// TwinCAT 3 PLC project MorpheePanel_PowerSupplyControl
// ProgramVersion: 3.1.4024.0
// libraries:
//   Tc2_Standard, * (Beckhoff Automation GmbH)
//   Tc2_System, * (Beckhoff Automation GmbH)
//   Tc3_Module, * (Beckhoff Automation GmbH)
// project tree:
//   DUTs/ panel302.TcDUT, RxData.TcDUT, TxData.TcDUT
//   GVLs/ GVL.TcGVL, GVL_Constant.TcGVL, GVL_Persistent.TcGVL, Safety_Tags.TcGVL
//   / PlcTask.TcTTO
//   POU/ DeviceManager.TcPOU, EthercatManager.TcPOU, GroupManager.TcPOU, Main.TcPOU, SafetyMgr.TcPOU, SetpointTest.TcPOU
// real-time tasks:
//   TASK PlcTask: cycle T#10ms, priority 20, ADS port 350
// I/O:
//   DEVICE Device 1 (EtherCAT), AmsNetId 5.146.184.42.2.1
//     Term 37 (EK1200) [EK1200-5000 EtherCAT Power supply (2A E-Bus)]
//       Term 2 (EL1819) [EL1819 16Ch. Dig. Input 24V, 10µs]
//       Term 3(EL6695) [EL6695 EtherCAT Bridge terminal (Primary)]
//       Term 4 (EK1521) [EK1521 1 port EtherCAT junction (FX-MultiMode)]
//         Term 5 (EK1501) [EK1501 EtherCAT Coupler (2A E-Bus, FX-MultiMode, ID switch)]
//           Term 6 (EL6070-0033) [EL6070-0033 1Ch. Licence key terminal, individual licences]
//           Term 7 (EL6910) [EL6910, TwinSAFE PLC]
//           Term 8 (EL1819) [EL1819 16Ch. Dig. Input 24V, 10µs]
//           Term 9 (EL1819) [EL1819 16Ch. Dig. Input 24V, 10µs]
//           Term 10 (EL1904) [EL1904, 4 Ch. Safety Input 24V, TwinSAFE]
//             modules: Module 1 (FSOES)
//           Term 11 (EL2809) [EL2809 16Ch. Dig. Output 24V, 0.5A]
//           Term 12 (EL2904) [EL2904, 4 Ch. Safety Output 24V, 0.5A, TwinSAFE]
//             modules: Module 1 (FSOES), Module 2 (DO)
//           Term 13 (EL2798) [EL2798 8Ch. Dig. Output 24V AC/DC, 2A, potential-free]
//           Term 14 (EL9410) [EL9410 E-Bus Power Supplier  (Diagnostics)]
//           Term 15 (EL3174) [EL3174 4Ch. Ana. Input +/-10V Diff., +/-20mA SingleEnded, 16 Bit]
//           Term 52 (EL6751) [EL6751 CANopen Master]
//           Term 53 (EL6751) [EL6751 CANopen Master]
//           Term 54 (EL6751) [EL6751 CANopen Master]
//           Term 20 (EK1122) [EK1122 2 port EtherCAT junction]
//             Box 22 (CX8110 EtherCAT slave) [CX8110 EtherCAT slave]
//       Term 3 (EK1122) [EK1122 2 port EtherCAT junction]
//         Term 48 (EK1100) [EK1100 EtherCAT Coupler (2A E-Bus)]
//           Term 49 (EL1819) [EL1819 16Ch. Dig. Input 24V, 10µs]
//           Term 50 (EL2809) [EL2809 16Ch. Dig. Output 24V, 0.5A]
//           Term 45 (EL1918) [EL1918, 8Ch. Safety Input 24V, TwinSAFE]
//             modules: Module 2 (FSLOGIC)
//           Term 52 (EL2904) [EL2904, 4 Ch. Safety Output 24V, 0.5A, TwinSAFE]
//             modules: Module 1 (FSOES), Module 2 (DO)
//           Term 60 (EL9011) [EL9011 End Terminal]
//         Term 54 (EK1100) [EK1100 EtherCAT Coupler (2A E-Bus)]
//           Term 55 (EL1819) [EL1819 16Ch. Dig. Input 24V, 10µs]
//           Term 56 (EL2809) [EL2809 16Ch. Dig. Output 24V, 0.5A]
//           Term 57 (EL1918) [EL1918, 8Ch. Safety Input 24V, TwinSAFE]
//             modules: Module 1 (FSOE), Module 2 (FSLOGIC)
//           Term 58 (EL2904) [EL2904, 4 Ch. Safety Output 24V, 0.5A, TwinSAFE]
//             modules: Module 1 (FSOES), Module 2 (DO)
//           Term 61 (EL9011) [EL9011 End Terminal]
//   DEVICE Device 6 (EL6751), AmsNetId 5.146.184.42.7.1
//     BIC2200_ID0
//     BIC2200_ID1
//     BIC2200_ID2
//     BIC2200_ID3
//     BIC2200_ID4
//     BIC2200_ID5
//     BIC2200_ID6
//     BIC2200_ID7
//   DEVICE Device 7 (EL6751), AmsNetId 5.146.184.42.8.1
//     BIC2200_ID0
//     BIC2200_ID1
//     BIC2200_ID2
//     BIC2200_ID3
//     BIC2200_ID4
//     BIC2200_ID5
//     BIC2200_ID6
//     BIC2200_ID7
//   DEVICE Device 5 (EL6751), AmsNetId 5.146.184.42.6.1
//     DPU3200_ID3
//     DPU3200_ID5
//     DPU3200_ID6
//     DPU3200_ID7
//   DEVICE Device 2 (EtherCAT Automation Protocol), AmsNetId 5.146.184.42.3.1
//     Box 43 (Publisher)
//     Box 44 (Subscriber)
//   DEVICE Device 10 (EtherCAT Slave), AmsNetId 5.146.184.42.11.255
// variable links:
//   Device 1 (EtherCAT) <-> Device 1 (EtherCAT)/Term 37 (EK1200)/Term 3 (EK1122)/Term 48 (EK1100)/Term 45 (EL1918)
//     Term 37 (EK1200)/Term 3 (EK1122)/Term 54 (EK1100)/Term 57 (EL1918)/Module 1 (FSOE)/FSoE Inputs/FSOE <-> ConnectionOutputs/Message_7 RxPDO
//     Term 37 (EK1200)/Term 3 (EK1122)/Term 54 (EK1100)/Term 57 (EL1918)/Module 1 (FSOE)/FSoE Outputs/FSOE <-> ConnectionInputs/Message_7 TxPDO
//     Term 37 (EK1200)/Term 3 (EK1122)/Term 54 (EK1100)/Term 58 (EL2904)/Module 1 (FSOES)/RxPDO/FSOE <-> ConnectionInputs/Message_10 TxPDO
//     Term 37 (EK1200)/Term 4 (EK1521)/Term 5 (EK1501)/Term 10 (EL1904)/Module 1 (FSOES)/RxPDO/FSOE <-> ConnectionInputs/Message_12 TxPDO
//     Term 37 (EK1200)/Term 4 (EK1521)/Term 5 (EK1501)/Term 12 (EL2904)/Module 1 (FSOES)/RxPDO/FSOE <-> ConnectionInputs/Message_3 TxPDO
//     Term 37 (EK1200)/Term 4 (EK1521)/Term 5 (EK1501)/Term 12 (EL2904)/Module 1 (FSOES)/TxPDO/FSOE <-> ConnectionOutputs/Message_3 RxPDO
//   Device 1 (EtherCAT) <-> Device 1 (EtherCAT)/Term 37 (EK1200)/Term 3 (EK1122)/Term 48 (EK1100)/Term 52 (EL2904)
//     Term 37 (EK1200)/Term 3 (EK1122)/Term 48 (EK1100)/Term 45 (EL1918)/ConnectionInputs/Message_8 TxPDO <-> Module 1 (FSOES)/RxPDO/FSOE
//     Term 37 (EK1200)/Term 3 (EK1122)/Term 48 (EK1100)/Term 45 (EL1918)/ConnectionOutputs/Message_8 RxPDO <-> Module 1 (FSOES)/TxPDO/FSOE
//   Device 1 (EtherCAT) <-> Device 1 (EtherCAT)/Term 37 (EK1200)/Term 3 (EK1122)/Term 54 (EK1100)/Term 58 (EL2904)
//     Term 37 (EK1200)/Term 3 (EK1122)/Term 48 (EK1100)/Term 45 (EL1918)/ConnectionOutputs/Message_10 RxPDO <-> Module 1 (FSOES)/TxPDO/FSOE
//   Device 1 (EtherCAT) <-> Device 1 (EtherCAT)/Term 37 (EK1200)/Term 3(EL6695)
//     Term 37 (EK1200)/Term 4 (EK1521)/Term 5 (EK1501)/Term 20 (EK1122)/Box 22 (CX8110 EtherCAT slave)/IO Inputs/Pdo Entry 10 <-> IO Outputs/Pdo Entry 10
//     Term 37 (EK1200)/Term 4 (EK1521)/Term 5 (EK1501)/Term 20 (EK1122)/Box 22 (CX8110 EtherCAT slave)/IO Inputs/Pdo Entry 11 <-> IO Outputs/Pdo Entry 11
//     Term 37 (EK1200)/Term 4 (EK1521)/Term 5 (EK1501)/Term 20 (EK1122)/Box 22 (CX8110 EtherCAT slave)/IO Inputs/Pdo Entry 15 <-> IO Outputs/Pdo Entry 15
//     Term 37 (EK1200)/Term 4 (EK1521)/Term 5 (EK1501)/Term 20 (EK1122)/Box 22 (CX8110 EtherCAT slave)/IO Inputs/Pdo Entry 16 <-> IO Outputs/Pdo Entry 16
//     Term 37 (EK1200)/Term 4 (EK1521)/Term 5 (EK1501)/Term 20 (EK1122)/Box 22 (CX8110 EtherCAT slave)/IO Inputs/Pdo Entry 20 <-> IO Outputs/Pdo Entry 20
//     Term 37 (EK1200)/Term 4 (EK1521)/Term 5 (EK1501)/Term 20 (EK1122)/Box 22 (CX8110 EtherCAT slave)/IO Inputs/Pdo Entry 21 <-> IO Outputs/Pdo Entry 21
//     Term 37 (EK1200)/Term 4 (EK1521)/Term 5 (EK1501)/Term 20 (EK1122)/Box 22 (CX8110 EtherCAT slave)/IO Inputs/Pdo Entry 25 <-> IO Outputs/Pdo Entry 25
//     Term 37 (EK1200)/Term 4 (EK1521)/Term 5 (EK1501)/Term 20 (EK1122)/Box 22 (CX8110 EtherCAT slave)/IO Inputs/Pdo Entry 26 <-> IO Outputs/Pdo Entry 26
//     Term 37 (EK1200)/Term 4 (EK1521)/Term 5 (EK1501)/Term 20 (EK1122)/Box 22 (CX8110 EtherCAT slave)/IO Inputs/Pdo Entry 31 <-> IO Outputs/Pdo Entry 31
//     Term 37 (EK1200)/Term 4 (EK1521)/Term 5 (EK1501)/Term 20 (EK1122)/Box 22 (CX8110 EtherCAT slave)/IO Inputs/Pdo Entry 32 <-> IO Outputs/Pdo Entry 32
//     Term 37 (EK1200)/Term 4 (EK1521)/Term 5 (EK1501)/Term 20 (EK1122)/Box 22 (CX8110 EtherCAT slave)/IO Inputs/Pdo Entry 36 <-> IO Outputs/Pdo Entry 36
//     Term 37 (EK1200)/Term 4 (EK1521)/Term 5 (EK1501)/Term 20 (EK1122)/Box 22 (CX8110 EtherCAT slave)/IO Inputs/Pdo Entry 37 <-> IO Outputs/Pdo Entry 37
//     Term 37 (EK1200)/Term 4 (EK1521)/Term 5 (EK1501)/Term 20 (EK1122)/Box 22 (CX8110 EtherCAT slave)/IO Inputs/Pdo Entry 41 <-> IO Outputs/Pdo Entry 41
//     Term 37 (EK1200)/Term 4 (EK1521)/Term 5 (EK1501)/Term 20 (EK1122)/Box 22 (CX8110 EtherCAT slave)/IO Inputs/Pdo Entry 42 <-> IO Outputs/Pdo Entry 42
//     Term 37 (EK1200)/Term 4 (EK1521)/Term 5 (EK1501)/Term 20 (EK1122)/Box 22 (CX8110 EtherCAT slave)/IO Inputs/Pdo Entry 46 <-> IO Outputs/Pdo Entry 46
//     Term 37 (EK1200)/Term 4 (EK1521)/Term 5 (EK1501)/Term 20 (EK1122)/Box 22 (CX8110 EtherCAT slave)/IO Inputs/Pdo Entry 47 <-> IO Outputs/Pdo Entry 47
//     Term 37 (EK1200)/Term 4 (EK1521)/Term 5 (EK1501)/Term 20 (EK1122)/Box 22 (CX8110 EtherCAT slave)/IO Inputs/Pdo Entry 5 <-> IO Outputs/Pdo Entry 5
//     Term 37 (EK1200)/Term 4 (EK1521)/Term 5 (EK1501)/Term 20 (EK1122)/Box 22 (CX8110 EtherCAT slave)/IO Inputs/Pdo Entry 51 <-> IO Outputs/Pdo Entry 51
//     Term 37 (EK1200)/Term 4 (EK1521)/Term 5 (EK1501)/Term 20 (EK1122)/Box 22 (CX8110 EtherCAT slave)/IO Inputs/Pdo Entry 52 <-> IO Outputs/Pdo Entry 52
//     Term 37 (EK1200)/Term 4 (EK1521)/Term 5 (EK1501)/Term 20 (EK1122)/Box 22 (CX8110 EtherCAT slave)/IO Inputs/Pdo Entry 56 <-> IO Outputs/Pdo Entry 56
//     Term 37 (EK1200)/Term 4 (EK1521)/Term 5 (EK1501)/Term 20 (EK1122)/Box 22 (CX8110 EtherCAT slave)/IO Inputs/Pdo Entry 57 <-> IO Outputs/Pdo Entry 57
//     Term 37 (EK1200)/Term 4 (EK1521)/Term 5 (EK1501)/Term 20 (EK1122)/Box 22 (CX8110 EtherCAT slave)/IO Inputs/Pdo Entry 58 <-> IO Outputs/Pdo Entry 58
//     Term 37 (EK1200)/Term 4 (EK1521)/Term 5 (EK1501)/Term 20 (EK1122)/Box 22 (CX8110 EtherCAT slave)/IO Inputs/Pdo Entry 6 <-> IO Outputs/Pdo Entry 6
//     Term 37 (EK1200)/Term 4 (EK1521)/Term 5 (EK1501)/Term 20 (EK1122)/Box 22 (CX8110 EtherCAT slave)/IO Inputs/Pdo Entry 62 <-> IO Outputs/Pdo Entry 62
//     Term 37 (EK1200)/Term 4 (EK1521)/Term 5 (EK1501)/Term 20 (EK1122)/Box 22 (CX8110 EtherCAT slave)/IO Inputs/Pdo Entry 63 <-> IO Outputs/Pdo Entry 63
//     Term 37 (EK1200)/Term 4 (EK1521)/Term 5 (EK1501)/Term 20 (EK1122)/Box 22 (CX8110 EtherCAT slave)/IO Inputs/Pdo Entry 67 <-> IO Outputs/Pdo Entry 67
//     Term 37 (EK1200)/Term 4 (EK1521)/Term 5 (EK1501)/Term 20 (EK1122)/Box 22 (CX8110 EtherCAT slave)/IO Inputs/Pdo Entry 68 <-> IO Outputs/Pdo Entry 68
//     Term 37 (EK1200)/Term 4 (EK1521)/Term 5 (EK1501)/Term 20 (EK1122)/Box 22 (CX8110 EtherCAT slave)/IO Inputs/Pdo Entry 72 <-> IO Outputs/Pdo Entry 72
//     Term 37 (EK1200)/Term 4 (EK1521)/Term 5 (EK1501)/Term 20 (EK1122)/Box 22 (CX8110 EtherCAT slave)/IO Inputs/Pdo Entry 73 <-> IO Outputs/Pdo Entry 73
//     Term 37 (EK1200)/Term 4 (EK1521)/Term 5 (EK1501)/Term 20 (EK1122)/Box 22 (CX8110 EtherCAT slave)/IO Inputs/Pdo Entry 77 <-> IO Outputs/Pdo Entry 77
//     Term 37 (EK1200)/Term 4 (EK1521)/Term 5 (EK1501)/Term 20 (EK1122)/Box 22 (CX8110 EtherCAT slave)/IO Inputs/Pdo Entry 78 <-> IO Outputs/Pdo Entry 78
//     Term 37 (EK1200)/Term 4 (EK1521)/Term 5 (EK1501)/Term 20 (EK1122)/Box 22 (CX8110 EtherCAT slave)/IO Inputs/Pdo Entry 82 <-> IO Outputs/Pdo Entry 82
//     Term 37 (EK1200)/Term 4 (EK1521)/Term 5 (EK1501)/Term 20 (EK1122)/Box 22 (CX8110 EtherCAT slave)/IO Inputs/Pdo Entry 83 <-> IO Outputs/Pdo Entry 83
//     Term 37 (EK1200)/Term 4 (EK1521)/Term 5 (EK1501)/Term 20 (EK1122)/Box 22 (CX8110 EtherCAT slave)/IO Inputs/Pdo Entry 84 <-> IO Outputs/Pdo Entry 84
//     Term 37 (EK1200)/Term 4 (EK1521)/Term 5 (EK1501)/Term 20 (EK1122)/Box 22 (CX8110 EtherCAT slave)/IO Inputs/Pdo Entry 88 <-> IO Outputs/Pdo Entry 88
//     Term 37 (EK1200)/Term 4 (EK1521)/Term 5 (EK1501)/Term 20 (EK1122)/Box 22 (CX8110 EtherCAT slave)/IO Inputs/Pdo Entry 89 <-> IO Outputs/Pdo Entry 89
//     Term 37 (EK1200)/Term 4 (EK1521)/Term 5 (EK1501)/Term 20 (EK1122)/Box 22 (CX8110 EtherCAT slave)/IO Inputs/Pdo Entry 93 <-> IO Outputs/Pdo Entry 93
//     Term 37 (EK1200)/Term 4 (EK1521)/Term 5 (EK1501)/Term 20 (EK1122)/Box 22 (CX8110 EtherCAT slave)/IO Inputs/Pdo Entry 94 <-> IO Outputs/Pdo Entry 94
//     Term 37 (EK1200)/Term 4 (EK1521)/Term 5 (EK1501)/Term 20 (EK1122)/Box 22 (CX8110 EtherCAT slave)/IO Inputs/Pdo Entry 98 <-> IO Outputs/Pdo Entry 98
//     Term 37 (EK1200)/Term 4 (EK1521)/Term 5 (EK1501)/Term 20 (EK1122)/Box 22 (CX8110 EtherCAT slave)/IO Inputs/Pdo Entry 99 <-> IO Outputs/Pdo Entry 99
//     Term 37 (EK1200)/Term 4 (EK1521)/Term 5 (EK1501)/Term 20 (EK1122)/Box 22 (CX8110 EtherCAT slave)/IO Outputs/Pdo Entry 11 <-> IO Inputs/Pdo Entry 11
//     Term 37 (EK1200)/Term 4 (EK1521)/Term 5 (EK1501)/Term 20 (EK1122)/Box 22 (CX8110 EtherCAT slave)/IO Outputs/Pdo Entry 32 <-> IO Inputs/Pdo Entry 32
//     Term 37 (EK1200)/Term 4 (EK1521)/Term 5 (EK1501)/Term 20 (EK1122)/Box 22 (CX8110 EtherCAT slave)/IO Outputs/Pdo Entry 37 <-> IO Inputs/Pdo Entry 37
//     Term 37 (EK1200)/Term 4 (EK1521)/Term 5 (EK1501)/Term 20 (EK1122)/Box 22 (CX8110 EtherCAT slave)/IO Outputs/Pdo Entry 6 <-> IO Inputs/Pdo Entry 6
//     Term 37 (EK1200)/Term 4 (EK1521)/Term 5 (EK1501)/Term 20 (EK1122)/Box 22 (CX8110 EtherCAT slave)/IO Outputs/Pdo Entry 63 <-> IO Inputs/Pdo Entry 63
//     Term 37 (EK1200)/Term 4 (EK1521)/Term 5 (EK1501)/Term 20 (EK1122)/Box 22 (CX8110 EtherCAT slave)/IO Outputs/Pdo Entry 89 <-> IO Inputs/Pdo Entry 89
//   Device 1 (EtherCAT) <-> Device 1 (EtherCAT)/Term 37 (EK1200)/Term 4 (EK1521)/Term 5 (EK1501)/Term 10 (EL1904)
//     Term 37 (EK1200)/Term 3 (EK1122)/Term 48 (EK1100)/Term 45 (EL1918)/ConnectionOutputs/Message_12 RxPDO <-> Module 1 (FSOES)/TxPDO/FSOE
//   Device 1 (EtherCAT) <-> Device 1 (EtherCAT)/Term 37 (EK1200)/Term 4 (EK1521)/Term 5 (EK1501)/Term 20 (EK1122)/Box 22 (CX8110 EtherCAT slave)
//     Term 37 (EK1200)/Term 3(EL6695)/IO Inputs/Pdo Entry 1 <-> IO Outputs/Pdo Entry 1
//     Term 37 (EK1200)/Term 3(EL6695)/IO Inputs/Pdo Entry 10 <-> IO Outputs/Pdo Entry 10
//     Term 37 (EK1200)/Term 3(EL6695)/IO Inputs/Pdo Entry 12 <-> IO Outputs/Pdo Entry 12
//     Term 37 (EK1200)/Term 3(EL6695)/IO Inputs/Pdo Entry 13 <-> IO Outputs/Pdo Entry 13
//     Term 37 (EK1200)/Term 3(EL6695)/IO Inputs/Pdo Entry 14 <-> IO Outputs/Pdo Entry 14
//     Term 37 (EK1200)/Term 3(EL6695)/IO Inputs/Pdo Entry 15 <-> IO Outputs/Pdo Entry 15
//     Term 37 (EK1200)/Term 3(EL6695)/IO Inputs/Pdo Entry 16 <-> IO Outputs/Pdo Entry 16
//     Term 37 (EK1200)/Term 3(EL6695)/IO Inputs/Pdo Entry 17 <-> IO Outputs/Pdo Entry 17
//     Term 37 (EK1200)/Term 3(EL6695)/IO Inputs/Pdo Entry 18 <-> IO Outputs/Pdo Entry 18
//     Term 37 (EK1200)/Term 3(EL6695)/IO Inputs/Pdo Entry 19 <-> IO Outputs/Pdo Entry 19
//     Term 37 (EK1200)/Term 3(EL6695)/IO Inputs/Pdo Entry 2 <-> IO Outputs/Pdo Entry 2
//     Term 37 (EK1200)/Term 3(EL6695)/IO Inputs/Pdo Entry 20 <-> IO Outputs/Pdo Entry 20
//     Term 37 (EK1200)/Term 3(EL6695)/IO Inputs/Pdo Entry 21 <-> IO Outputs/Pdo Entry 21
//     Term 37 (EK1200)/Term 3(EL6695)/IO Inputs/Pdo Entry 22 <-> IO Outputs/Pdo Entry 22
//     Term 37 (EK1200)/Term 3(EL6695)/IO Inputs/Pdo Entry 23 <-> IO Outputs/Pdo Entry 23
//     Term 37 (EK1200)/Term 3(EL6695)/IO Inputs/Pdo Entry 24 <-> IO Outputs/Pdo Entry 24
//     Term 37 (EK1200)/Term 3(EL6695)/IO Inputs/Pdo Entry 25 <-> IO Outputs/Pdo Entry 25
//     Term 37 (EK1200)/Term 3(EL6695)/IO Inputs/Pdo Entry 26 <-> IO Outputs/Pdo Entry 26
//     Term 37 (EK1200)/Term 3(EL6695)/IO Inputs/Pdo Entry 27 <-> IO Outputs/Pdo Entry 27
//     Term 37 (EK1200)/Term 3(EL6695)/IO Inputs/Pdo Entry 28 <-> IO Outputs/Pdo Entry 28
//     Term 37 (EK1200)/Term 3(EL6695)/IO Inputs/Pdo Entry 29 <-> IO Outputs/Pdo Entry 29
//     Term 37 (EK1200)/Term 3(EL6695)/IO Inputs/Pdo Entry 3 <-> IO Outputs/Pdo Entry 3
//     Term 37 (EK1200)/Term 3(EL6695)/IO Inputs/Pdo Entry 30 <-> IO Outputs/Pdo Entry 30
//     Term 37 (EK1200)/Term 3(EL6695)/IO Inputs/Pdo Entry 31 <-> IO Outputs/Pdo Entry 31
//     Term 37 (EK1200)/Term 3(EL6695)/IO Inputs/Pdo Entry 33 <-> IO Outputs/Pdo Entry 33
//     Term 37 (EK1200)/Term 3(EL6695)/IO Inputs/Pdo Entry 34 <-> IO Outputs/Pdo Entry 34
//     Term 37 (EK1200)/Term 3(EL6695)/IO Inputs/Pdo Entry 35 <-> IO Outputs/Pdo Entry 35
//     Term 37 (EK1200)/Term 3(EL6695)/IO Inputs/Pdo Entry 36 <-> IO Outputs/Pdo Entry 36
//     Term 37 (EK1200)/Term 3(EL6695)/IO Inputs/Pdo Entry 38 <-> IO Outputs/Pdo Entry 38
//     Term 37 (EK1200)/Term 3(EL6695)/IO Inputs/Pdo Entry 39 <-> IO Outputs/Pdo Entry 39
//     Term 37 (EK1200)/Term 3(EL6695)/IO Inputs/Pdo Entry 4 <-> IO Outputs/Pdo Entry 4
//     Term 37 (EK1200)/Term 3(EL6695)/IO Inputs/Pdo Entry 40 <-> IO Outputs/Pdo Entry 40
//     Term 37 (EK1200)/Term 3(EL6695)/IO Inputs/Pdo Entry 41 <-> IO Outputs/Pdo Entry 41
//     Term 37 (EK1200)/Term 3(EL6695)/IO Inputs/Pdo Entry 42 <-> IO Outputs/Pdo Entry 42
//     Term 37 (EK1200)/Term 3(EL6695)/IO Inputs/Pdo Entry 43 <-> IO Outputs/Pdo Entry 43
//     Term 37 (EK1200)/Term 3(EL6695)/IO Inputs/Pdo Entry 44 <-> IO Outputs/Pdo Entry 44
//     Term 37 (EK1200)/Term 3(EL6695)/IO Inputs/Pdo Entry 45 <-> IO Outputs/Pdo Entry 45
//     Term 37 (EK1200)/Term 3(EL6695)/IO Inputs/Pdo Entry 46 <-> IO Outputs/Pdo Entry 46
//     Term 37 (EK1200)/Term 3(EL6695)/IO Inputs/Pdo Entry 47 <-> IO Outputs/Pdo Entry 47
//     Term 37 (EK1200)/Term 3(EL6695)/IO Inputs/Pdo Entry 48 <-> IO Outputs/Pdo Entry 48
//     Term 37 (EK1200)/Term 3(EL6695)/IO Inputs/Pdo Entry 49 <-> IO Outputs/Pdo Entry 49
//     Term 37 (EK1200)/Term 3(EL6695)/IO Inputs/Pdo Entry 5 <-> IO Outputs/Pdo Entry 5
//     Term 37 (EK1200)/Term 3(EL6695)/IO Inputs/Pdo Entry 50 <-> IO Outputs/Pdo Entry 50
//     Term 37 (EK1200)/Term 3(EL6695)/IO Inputs/Pdo Entry 51 <-> IO Outputs/Pdo Entry 51
//     Term 37 (EK1200)/Term 3(EL6695)/IO Inputs/Pdo Entry 52 <-> IO Outputs/Pdo Entry 52
//     Term 37 (EK1200)/Term 3(EL6695)/IO Inputs/Pdo Entry 53 <-> IO Outputs/Pdo Entry 53
//     Term 37 (EK1200)/Term 3(EL6695)/IO Inputs/Pdo Entry 54 <-> IO Outputs/Pdo Entry 54
//     Term 37 (EK1200)/Term 3(EL6695)/IO Inputs/Pdo Entry 55 <-> IO Outputs/Pdo Entry 55
//     Term 37 (EK1200)/Term 3(EL6695)/IO Inputs/Pdo Entry 56 <-> IO Outputs/Pdo Entry 56
//     Term 37 (EK1200)/Term 3(EL6695)/IO Inputs/Pdo Entry 57 <-> IO Outputs/Pdo Entry 57
//     Term 37 (EK1200)/Term 3(EL6695)/IO Inputs/Pdo Entry 58 <-> IO Outputs/Pdo Entry 58
//     Term 37 (EK1200)/Term 3(EL6695)/IO Inputs/Pdo Entry 59 <-> IO Outputs/Pdo Entry 59
//     Term 37 (EK1200)/Term 3(EL6695)/IO Inputs/Pdo Entry 60 <-> IO Outputs/Pdo Entry 60
//     Term 37 (EK1200)/Term 3(EL6695)/IO Inputs/Pdo Entry 61 <-> IO Outputs/Pdo Entry 61
//     Term 37 (EK1200)/Term 3(EL6695)/IO Inputs/Pdo Entry 62 <-> IO Outputs/Pdo Entry 62
//     Term 37 (EK1200)/Term 3(EL6695)/IO Inputs/Pdo Entry 64 <-> IO Outputs/Pdo Entry 64
//     Term 37 (EK1200)/Term 3(EL6695)/IO Inputs/Pdo Entry 65 <-> IO Outputs/Pdo Entry 65
//     Term 37 (EK1200)/Term 3(EL6695)/IO Inputs/Pdo Entry 66 <-> IO Outputs/Pdo Entry 66
//     Term 37 (EK1200)/Term 3(EL6695)/IO Inputs/Pdo Entry 67 <-> IO Outputs/Pdo Entry 67
//     Term 37 (EK1200)/Term 3(EL6695)/IO Inputs/Pdo Entry 68 <-> IO Outputs/Pdo Entry 68
//     Term 37 (EK1200)/Term 3(EL6695)/IO Inputs/Pdo Entry 69 <-> IO Outputs/Pdo Entry 69
//     Term 37 (EK1200)/Term 3(EL6695)/IO Inputs/Pdo Entry 7 <-> IO Outputs/Pdo Entry 7
//     Term 37 (EK1200)/Term 3(EL6695)/IO Inputs/Pdo Entry 70 <-> IO Outputs/Pdo Entry 70
//     Term 37 (EK1200)/Term 3(EL6695)/IO Inputs/Pdo Entry 71 <-> IO Outputs/Pdo Entry 71
//     Term 37 (EK1200)/Term 3(EL6695)/IO Inputs/Pdo Entry 72 <-> IO Outputs/Pdo Entry 72
//     Term 37 (EK1200)/Term 3(EL6695)/IO Inputs/Pdo Entry 73 <-> IO Outputs/Pdo Entry 73
//     Term 37 (EK1200)/Term 3(EL6695)/IO Inputs/Pdo Entry 74 <-> IO Outputs/Pdo Entry 74
//     Term 37 (EK1200)/Term 3(EL6695)/IO Inputs/Pdo Entry 75 <-> IO Outputs/Pdo Entry 75
//     Term 37 (EK1200)/Term 3(EL6695)/IO Inputs/Pdo Entry 76 <-> IO Outputs/Pdo Entry 76
//     Term 37 (EK1200)/Term 3(EL6695)/IO Inputs/Pdo Entry 77 <-> IO Outputs/Pdo Entry 77
//     Term 37 (EK1200)/Term 3(EL6695)/IO Inputs/Pdo Entry 78 <-> IO Outputs/Pdo Entry 78
//     Term 37 (EK1200)/Term 3(EL6695)/IO Inputs/Pdo Entry 79 <-> IO Outputs/Pdo Entry 79
//     Term 37 (EK1200)/Term 3(EL6695)/IO Inputs/Pdo Entry 8 <-> IO Outputs/Pdo Entry 8
//     Term 37 (EK1200)/Term 3(EL6695)/IO Inputs/Pdo Entry 80 <-> IO Outputs/Pdo Entry 80
//     Term 37 (EK1200)/Term 3(EL6695)/IO Inputs/Pdo Entry 81 <-> IO Outputs/Pdo Entry 81
//     Term 37 (EK1200)/Term 3(EL6695)/IO Inputs/Pdo Entry 82 <-> IO Outputs/Pdo Entry 82
//     Term 37 (EK1200)/Term 3(EL6695)/IO Inputs/Pdo Entry 83 <-> IO Outputs/Pdo Entry 83
//     Term 37 (EK1200)/Term 3(EL6695)/IO Inputs/Pdo Entry 84 <-> IO Outputs/Pdo Entry 84
//     Term 37 (EK1200)/Term 3(EL6695)/IO Inputs/Pdo Entry 85 <-> IO Outputs/Pdo Entry 85
//     Term 37 (EK1200)/Term 3(EL6695)/IO Inputs/Pdo Entry 86 <-> IO Outputs/Pdo Entry 86
//     Term 37 (EK1200)/Term 3(EL6695)/IO Inputs/Pdo Entry 87 <-> IO Outputs/Pdo Entry 87
//     Term 37 (EK1200)/Term 3(EL6695)/IO Inputs/Pdo Entry 88 <-> IO Outputs/Pdo Entry 88
//     Term 37 (EK1200)/Term 3(EL6695)/IO Inputs/Pdo Entry 9 <-> IO Outputs/Pdo Entry 9
//     Term 37 (EK1200)/Term 3(EL6695)/IO Inputs/Pdo Entry 90 <-> IO Outputs/Pdo Entry 90
//     Term 37 (EK1200)/Term 3(EL6695)/IO Outputs/Pdo Entry 1 <-> IO Inputs/Pdo Entry 1
//     Term 37 (EK1200)/Term 3(EL6695)/IO Outputs/Pdo Entry 100 <-> IO Inputs/Pdo Entry 100
//     Term 37 (EK1200)/Term 3(EL6695)/IO Outputs/Pdo Entry 101 <-> IO Inputs/Pdo Entry 101
//     Term 37 (EK1200)/Term 3(EL6695)/IO Outputs/Pdo Entry 102 <-> IO Inputs/Pdo Entry 102
//     Term 37 (EK1200)/Term 3(EL6695)/IO Outputs/Pdo Entry 12 <-> IO Inputs/Pdo Entry 12
//     Term 37 (EK1200)/Term 3(EL6695)/IO Outputs/Pdo Entry 13 <-> IO Inputs/Pdo Entry 13
//     Term 37 (EK1200)/Term 3(EL6695)/IO Outputs/Pdo Entry 14 <-> IO Inputs/Pdo Entry 14
//     Term 37 (EK1200)/Term 3(EL6695)/IO Outputs/Pdo Entry 17 <-> IO Inputs/Pdo Entry 17
//     Term 37 (EK1200)/Term 3(EL6695)/IO Outputs/Pdo Entry 18 <-> IO Inputs/Pdo Entry 18
//     Term 37 (EK1200)/Term 3(EL6695)/IO Outputs/Pdo Entry 19 <-> IO Inputs/Pdo Entry 19
//     Term 37 (EK1200)/Term 3(EL6695)/IO Outputs/Pdo Entry 2 <-> IO Inputs/Pdo Entry 2
//     Term 37 (EK1200)/Term 3(EL6695)/IO Outputs/Pdo Entry 22 <-> IO Inputs/Pdo Entry 22
//     Term 37 (EK1200)/Term 3(EL6695)/IO Outputs/Pdo Entry 23 <-> IO Inputs/Pdo Entry 23
//     Term 37 (EK1200)/Term 3(EL6695)/IO Outputs/Pdo Entry 24 <-> IO Inputs/Pdo Entry 24
//     Term 37 (EK1200)/Term 3(EL6695)/IO Outputs/Pdo Entry 27 <-> IO Inputs/Pdo Entry 27
//     Term 37 (EK1200)/Term 3(EL6695)/IO Outputs/Pdo Entry 28 <-> IO Inputs/Pdo Entry 28
//     Term 37 (EK1200)/Term 3(EL6695)/IO Outputs/Pdo Entry 29 <-> IO Inputs/Pdo Entry 29
//     Term 37 (EK1200)/Term 3(EL6695)/IO Outputs/Pdo Entry 3 <-> IO Inputs/Pdo Entry 3
//     Term 37 (EK1200)/Term 3(EL6695)/IO Outputs/Pdo Entry 30 <-> IO Inputs/Pdo Entry 30
//     Term 37 (EK1200)/Term 3(EL6695)/IO Outputs/Pdo Entry 33 <-> IO Inputs/Pdo Entry 33
//     Term 37 (EK1200)/Term 3(EL6695)/IO Outputs/Pdo Entry 34 <-> IO Inputs/Pdo Entry 34
//     Term 37 (EK1200)/Term 3(EL6695)/IO Outputs/Pdo Entry 35 <-> IO Inputs/Pdo Entry 35
//     Term 37 (EK1200)/Term 3(EL6695)/IO Outputs/Pdo Entry 38 <-> IO Inputs/Pdo Entry 38
//     Term 37 (EK1200)/Term 3(EL6695)/IO Outputs/Pdo Entry 39 <-> IO Inputs/Pdo Entry 39
//     Term 37 (EK1200)/Term 3(EL6695)/IO Outputs/Pdo Entry 4 <-> IO Inputs/Pdo Entry 4
//     Term 37 (EK1200)/Term 3(EL6695)/IO Outputs/Pdo Entry 40 <-> IO Inputs/Pdo Entry 40
//     Term 37 (EK1200)/Term 3(EL6695)/IO Outputs/Pdo Entry 43 <-> IO Inputs/Pdo Entry 43
//     Term 37 (EK1200)/Term 3(EL6695)/IO Outputs/Pdo Entry 44 <-> IO Inputs/Pdo Entry 44
//     Term 37 (EK1200)/Term 3(EL6695)/IO Outputs/Pdo Entry 45 <-> IO Inputs/Pdo Entry 45
//     Term 37 (EK1200)/Term 3(EL6695)/IO Outputs/Pdo Entry 48 <-> IO Inputs/Pdo Entry 48
//     Term 37 (EK1200)/Term 3(EL6695)/IO Outputs/Pdo Entry 49 <-> IO Inputs/Pdo Entry 49
//     Term 37 (EK1200)/Term 3(EL6695)/IO Outputs/Pdo Entry 50 <-> IO Inputs/Pdo Entry 50
//     Term 37 (EK1200)/Term 3(EL6695)/IO Outputs/Pdo Entry 53 <-> IO Inputs/Pdo Entry 53
//     Term 37 (EK1200)/Term 3(EL6695)/IO Outputs/Pdo Entry 54 <-> IO Inputs/Pdo Entry 54
//     Term 37 (EK1200)/Term 3(EL6695)/IO Outputs/Pdo Entry 55 <-> IO Inputs/Pdo Entry 55
//     Term 37 (EK1200)/Term 3(EL6695)/IO Outputs/Pdo Entry 59 <-> IO Inputs/Pdo Entry 59
//     Term 37 (EK1200)/Term 3(EL6695)/IO Outputs/Pdo Entry 60 <-> IO Inputs/Pdo Entry 60
//     Term 37 (EK1200)/Term 3(EL6695)/IO Outputs/Pdo Entry 61 <-> IO Inputs/Pdo Entry 61
//     Term 37 (EK1200)/Term 3(EL6695)/IO Outputs/Pdo Entry 64 <-> IO Inputs/Pdo Entry 64
//     Term 37 (EK1200)/Term 3(EL6695)/IO Outputs/Pdo Entry 65 <-> IO Inputs/Pdo Entry 65
//     Term 37 (EK1200)/Term 3(EL6695)/IO Outputs/Pdo Entry 66 <-> IO Inputs/Pdo Entry 66
//     Term 37 (EK1200)/Term 3(EL6695)/IO Outputs/Pdo Entry 69 <-> IO Inputs/Pdo Entry 69
//     Term 37 (EK1200)/Term 3(EL6695)/IO Outputs/Pdo Entry 7 <-> IO Inputs/Pdo Entry 7
//     Term 37 (EK1200)/Term 3(EL6695)/IO Outputs/Pdo Entry 70 <-> IO Inputs/Pdo Entry 70
//     Term 37 (EK1200)/Term 3(EL6695)/IO Outputs/Pdo Entry 71 <-> IO Inputs/Pdo Entry 71
//     Term 37 (EK1200)/Term 3(EL6695)/IO Outputs/Pdo Entry 74 <-> IO Inputs/Pdo Entry 74
//     Term 37 (EK1200)/Term 3(EL6695)/IO Outputs/Pdo Entry 75 <-> IO Inputs/Pdo Entry 75
//     Term 37 (EK1200)/Term 3(EL6695)/IO Outputs/Pdo Entry 76 <-> IO Inputs/Pdo Entry 76
//     Term 37 (EK1200)/Term 3(EL6695)/IO Outputs/Pdo Entry 79 <-> IO Inputs/Pdo Entry 79
//     Term 37 (EK1200)/Term 3(EL6695)/IO Outputs/Pdo Entry 8 <-> IO Inputs/Pdo Entry 8
//     Term 37 (EK1200)/Term 3(EL6695)/IO Outputs/Pdo Entry 80 <-> IO Inputs/Pdo Entry 80
//     Term 37 (EK1200)/Term 3(EL6695)/IO Outputs/Pdo Entry 81 <-> IO Inputs/Pdo Entry 81
//     Term 37 (EK1200)/Term 3(EL6695)/IO Outputs/Pdo Entry 85 <-> IO Inputs/Pdo Entry 85
//     Term 37 (EK1200)/Term 3(EL6695)/IO Outputs/Pdo Entry 86 <-> IO Inputs/Pdo Entry 86
//     Term 37 (EK1200)/Term 3(EL6695)/IO Outputs/Pdo Entry 87 <-> IO Inputs/Pdo Entry 87
//     Term 37 (EK1200)/Term 3(EL6695)/IO Outputs/Pdo Entry 9 <-> IO Inputs/Pdo Entry 9
//     Term 37 (EK1200)/Term 3(EL6695)/IO Outputs/Pdo Entry 90 <-> IO Inputs/Pdo Entry 90
//     Term 37 (EK1200)/Term 3(EL6695)/IO Outputs/Pdo Entry 91 <-> IO Inputs/Pdo Entry 91
//     Term 37 (EK1200)/Term 3(EL6695)/IO Outputs/Pdo Entry 92 <-> IO Inputs/Pdo Entry 92
//     Term 37 (EK1200)/Term 3(EL6695)/IO Outputs/Pdo Entry 95 <-> IO Inputs/Pdo Entry 95
//     Term 37 (EK1200)/Term 3(EL6695)/IO Outputs/Pdo Entry 96 <-> IO Inputs/Pdo Entry 96
//     Term 37 (EK1200)/Term 3(EL6695)/IO Outputs/Pdo Entry 97 <-> IO Inputs/Pdo Entry 97
//   MorpheePanel_PowerSupplyControl/MorpheePanel_PowerSupplyControl Instance <-> Device 1 (EtherCAT)/Term 37 (EK1200)/Term 3 (EK1122)/Term 48 (EK1100)/Term 45 (EL1918)
//     PlcTask Outputs/Safety_Tags.Reset <-> StandardOutputs/Standard In Var 1
//     PlcTask Outputs/Safety_Tags.Run <-> StandardOutputs/Standard In Var 9
//   MorpheePanel_PowerSupplyControl/MorpheePanel_PowerSupplyControl Instance <-> Device 1 (EtherCAT)/Term 37 (EK1200)/Term 3 (EK1122)/Term 48 (EK1100)/Term 50 (EL2809)
//     PlcTask Outputs/GVL.EL2809_Output[2,{0..15}] <-> Channel {1..16}/Output  (16 links)
//   MorpheePanel_PowerSupplyControl/MorpheePanel_PowerSupplyControl Instance <-> Device 1 (EtherCAT)/Term 37 (EK1200)/Term 3 (EK1122)/Term 54 (EK1100)/Term 56 (EL2809)
//     PlcTask Outputs/GVL.EL2809_Output[1,{0..15}] <-> Channel {1..16}/Output  (16 links)
//   MorpheePanel_PowerSupplyControl/MorpheePanel_PowerSupplyControl Instance <-> Device 1 (EtherCAT)/Term 37 (EK1200)/Term 4 (EK1521)/Term 5 (EK1501)/Term 11 (EL2809)
//     PlcTask Outputs/GVL.EL2809_Output[0,{0..15}] <-> Channel {1..16}/Output  (16 links)
//   MorpheePanel_PowerSupplyControl/MorpheePanel_PowerSupplyControl Instance <-> Device 1 (EtherCAT)/Term 37 (EK1200)/Term 4 (EK1521)/Term 5 (EK1501)/Term 13 (EL2798)
//     PlcTask Outputs/GVL.EL2798_Output[{0..3}] <-> Channel {1..4}/Output  (4 links)
//   MorpheePanel_PowerSupplyControl/MorpheePanel_PowerSupplyControl Instance <-> Device 1 (EtherCAT)/Term 37 (EK1200)/Term 4 (EK1521)/Term 5 (EK1501)/Term 15 (EL3174)
//     PlcTask Inputs/GVL.EL3174_Channel1_Value <-> AI Standard Channel 1/Value
//   MorpheePanel_PowerSupplyControl/MorpheePanel_PowerSupplyControl Instance <-> Device 1 (EtherCAT)/Term 37 (EK1200)/Term 4 (EK1521)/Term 5 (EK1501)/Term 8 (EL1819)
//     PlcTask Inputs/GVL.TemperatureFaultHigh[{0..10}] <-> Channel {1..11}/Input  (11 links)
//   MorpheePanel_PowerSupplyControl/MorpheePanel_PowerSupplyControl Instance <-> Device 1 (EtherCAT)/Term 37 (EK1200)/Term 4 (EK1521)/Term 5 (EK1501)/Term 9 (EL1819)
//     PlcTask Inputs/GVL.TemperatureFaultHigh[{11..19}] <-> Channel {1..9}/Input  (9 links)
//   MorpheePanel_PowerSupplyControl/MorpheePanel_PowerSupplyControl Instance <-> Device 10 (EtherCAT Slave)
//     PlcTask Inputs/GVL.NumericInput <-> Inputs/NumericInput_0
//     PlcTask Inputs/GVL.NumericInput @bit {16..3824 step 16} <-> Inputs/NumericInput_{1..239}  (239 links)
//     PlcTask Outputs/GVL.NumericOutput[0] <-> Outputs/dNumericOutput_0
//     PlcTask Outputs/GVL.NumericOutput[100] <-> Outputs/dNumericOutput_100
//     PlcTask Outputs/GVL.NumericOutput[101] <-> Outputs/dNumericOutput_101
//     PlcTask Outputs/GVL.NumericOutput[102] <-> Outputs/dNumericOutput_102
//     PlcTask Outputs/GVL.NumericOutput[103] <-> Outputs/dNumericOutput_103
//     PlcTask Outputs/GVL.NumericOutput[104] <-> Outputs/dNumericOutput_104
//     PlcTask Outputs/GVL.NumericOutput[105] <-> Outputs/dNumericOutput_105
//     PlcTask Outputs/GVL.NumericOutput[106] <-> Outputs/dNumericOutput_106
//     PlcTask Outputs/GVL.NumericOutput[107] <-> Outputs/dNumericOutput_107
//     PlcTask Outputs/GVL.NumericOutput[108] <-> Outputs/dNumericOutput_108
//     PlcTask Outputs/GVL.NumericOutput[109] <-> Outputs/dNumericOutput_109
//     PlcTask Outputs/GVL.NumericOutput[10] <-> Outputs/dNumericOutput_10
//     PlcTask Outputs/GVL.NumericOutput[110] <-> Outputs/dNumericOutput_110
//     PlcTask Outputs/GVL.NumericOutput[111] <-> Outputs/dNumericOutput_111
//     PlcTask Outputs/GVL.NumericOutput[112] <-> Outputs/dNumericOutput_112
//     PlcTask Outputs/GVL.NumericOutput[113] <-> Outputs/dNumericOutput_113
//     PlcTask Outputs/GVL.NumericOutput[114] <-> Outputs/dNumericOutput_114
//     PlcTask Outputs/GVL.NumericOutput[115] <-> Outputs/dNumericOutput_115
//     PlcTask Outputs/GVL.NumericOutput[116] <-> Outputs/dNumericOutput_116
//     PlcTask Outputs/GVL.NumericOutput[117] <-> Outputs/dNumericOutput_117
//     PlcTask Outputs/GVL.NumericOutput[118] <-> Outputs/dNumericOutput_118
//     PlcTask Outputs/GVL.NumericOutput[119] <-> Outputs/dNumericOutput_119
//     PlcTask Outputs/GVL.NumericOutput[11] <-> Outputs/dNumericOutput_11
//     PlcTask Outputs/GVL.NumericOutput[12] <-> Outputs/dNumericOutput_12
//     PlcTask Outputs/GVL.NumericOutput[13] <-> Outputs/dNumericOutput_13
//     PlcTask Outputs/GVL.NumericOutput[14] <-> Outputs/dNumericOutput_14
//     PlcTask Outputs/GVL.NumericOutput[15] <-> Outputs/dNumericOutput_15
//     PlcTask Outputs/GVL.NumericOutput[16] <-> Outputs/dNumericOutput_16
//     PlcTask Outputs/GVL.NumericOutput[17] <-> Outputs/dNumericOutput_17
//     PlcTask Outputs/GVL.NumericOutput[18] <-> Outputs/dNumericOutput_18
//     PlcTask Outputs/GVL.NumericOutput[19] <-> Outputs/dNumericOutput_19
//     PlcTask Outputs/GVL.NumericOutput[1] <-> Outputs/dNumericOutput_1
//     PlcTask Outputs/GVL.NumericOutput[20] <-> Outputs/dNumericOutput_20
//     PlcTask Outputs/GVL.NumericOutput[21] <-> Outputs/dNumericOutput_21
//     PlcTask Outputs/GVL.NumericOutput[22] <-> Outputs/dNumericOutput_22
//     PlcTask Outputs/GVL.NumericOutput[23] <-> Outputs/dNumericOutput_23
//     PlcTask Outputs/GVL.NumericOutput[24] <-> Outputs/dNumericOutput_24
//     PlcTask Outputs/GVL.NumericOutput[25] <-> Outputs/dNumericOutput_25
//     PlcTask Outputs/GVL.NumericOutput[26] <-> Outputs/dNumericOutput_26
//     PlcTask Outputs/GVL.NumericOutput[27] <-> Outputs/dNumericOutput_27
//     PlcTask Outputs/GVL.NumericOutput[28] <-> Outputs/dNumericOutput_28
//     PlcTask Outputs/GVL.NumericOutput[29] <-> Outputs/dNumericOutput_29
//     PlcTask Outputs/GVL.NumericOutput[2] <-> Outputs/dNumericOutput_2
//     PlcTask Outputs/GVL.NumericOutput[30] <-> Outputs/dNumericOutput_30
//     PlcTask Outputs/GVL.NumericOutput[31] <-> Outputs/dNumericOutput_31
//     PlcTask Outputs/GVL.NumericOutput[32] <-> Outputs/dNumericOutput_32
//     PlcTask Outputs/GVL.NumericOutput[33] <-> Outputs/dNumericOutput_33
//     PlcTask Outputs/GVL.NumericOutput[34] <-> Outputs/dNumericOutput_34
//     PlcTask Outputs/GVL.NumericOutput[35] <-> Outputs/dNumericOutput_35
//     PlcTask Outputs/GVL.NumericOutput[36] <-> Outputs/dNumericOutput_36
//     PlcTask Outputs/GVL.NumericOutput[37] <-> Outputs/dNumericOutput_37
//     PlcTask Outputs/GVL.NumericOutput[38] <-> Outputs/dNumericOutput_38
//     PlcTask Outputs/GVL.NumericOutput[39] <-> Outputs/dNumericOutput_39
//     PlcTask Outputs/GVL.NumericOutput[3] <-> Outputs/dNumericOutput_3
//     PlcTask Outputs/GVL.NumericOutput[40] <-> Outputs/dNumericOutput_40
//     PlcTask Outputs/GVL.NumericOutput[41] <-> Outputs/dNumericOutput_41
//     PlcTask Outputs/GVL.NumericOutput[42] <-> Outputs/dNumericOutput_42
//     PlcTask Outputs/GVL.NumericOutput[43] <-> Outputs/dNumericOutput_43
//     PlcTask Outputs/GVL.NumericOutput[44] <-> Outputs/dNumericOutput_44
//     PlcTask Outputs/GVL.NumericOutput[45] <-> Outputs/dNumericOutput_45
//     PlcTask Outputs/GVL.NumericOutput[46] <-> Outputs/dNumericOutput_46
//     PlcTask Outputs/GVL.NumericOutput[47] <-> Outputs/dNumericOutput_47
//     PlcTask Outputs/GVL.NumericOutput[48] <-> Outputs/dNumericOutput_48
//     PlcTask Outputs/GVL.NumericOutput[49] <-> Outputs/dNumericOutput_49
//     PlcTask Outputs/GVL.NumericOutput[4] <-> Outputs/dNumericOutput_4
//     PlcTask Outputs/GVL.NumericOutput[50] <-> Outputs/dNumericOutput_50
//     PlcTask Outputs/GVL.NumericOutput[51] <-> Outputs/dNumericOutput_51
//     PlcTask Outputs/GVL.NumericOutput[52] <-> Outputs/dNumericOutput_52
//     PlcTask Outputs/GVL.NumericOutput[53] <-> Outputs/dNumericOutput_53
//     PlcTask Outputs/GVL.NumericOutput[54] <-> Outputs/dNumericOutput_54
//     PlcTask Outputs/GVL.NumericOutput[55] <-> Outputs/dNumericOutput_55
//     PlcTask Outputs/GVL.NumericOutput[56] <-> Outputs/dNumericOutput_56
//     PlcTask Outputs/GVL.NumericOutput[57] <-> Outputs/dNumericOutput_57
//     PlcTask Outputs/GVL.NumericOutput[58] <-> Outputs/dNumericOutput_58
//     PlcTask Outputs/GVL.NumericOutput[59] <-> Outputs/dNumericOutput_59
//     PlcTask Outputs/GVL.NumericOutput[5] <-> Outputs/dNumericOutput_5
//     PlcTask Outputs/GVL.NumericOutput[60] <-> Outputs/dNumericOutput_60
//     PlcTask Outputs/GVL.NumericOutput[61] <-> Outputs/dNumericOutput_61
//     PlcTask Outputs/GVL.NumericOutput[62] <-> Outputs/dNumericOutput_62
//     PlcTask Outputs/GVL.NumericOutput[63] <-> Outputs/dNumericOutput_63
//     PlcTask Outputs/GVL.NumericOutput[64] <-> Outputs/dNumericOutput_64
//     PlcTask Outputs/GVL.NumericOutput[65] <-> Outputs/dNumericOutput_65
//     PlcTask Outputs/GVL.NumericOutput[66] <-> Outputs/dNumericOutput_66
//     PlcTask Outputs/GVL.NumericOutput[67] <-> Outputs/dNumericOutput_67
//     PlcTask Outputs/GVL.NumericOutput[68] <-> Outputs/dNumericOutput_68
//     PlcTask Outputs/GVL.NumericOutput[6] <-> Outputs/dNumericOutput_6
//     PlcTask Outputs/GVL.NumericOutput[70] <-> Outputs/dNumericOutput_70
//     PlcTask Outputs/GVL.NumericOutput[71] <-> Outputs/dNumericOutput_71
//     PlcTask Outputs/GVL.NumericOutput[72] <-> Outputs/dNumericOutput_72
//     PlcTask Outputs/GVL.NumericOutput[73] <-> Outputs/dNumericOutput_73
//     PlcTask Outputs/GVL.NumericOutput[74] <-> Outputs/dNumericOutput_74
//     PlcTask Outputs/GVL.NumericOutput[75] <-> Outputs/dNumericOutput_75
//     PlcTask Outputs/GVL.NumericOutput[76] <-> Outputs/dNumericOutput_76
//     PlcTask Outputs/GVL.NumericOutput[77] <-> Outputs/dNumericOutput_77
//     PlcTask Outputs/GVL.NumericOutput[78] <-> Outputs/dNumericOutput_78
//     PlcTask Outputs/GVL.NumericOutput[79] <-> Outputs/dNumericOutput_79
//     PlcTask Outputs/GVL.NumericOutput[7] <-> Outputs/dNumericOutput_7
//     PlcTask Outputs/GVL.NumericOutput[80] <-> Outputs/dNumericOutput_80
//     PlcTask Outputs/GVL.NumericOutput[81] <-> Outputs/dNumericOutput_81
//     PlcTask Outputs/GVL.NumericOutput[82] <-> Outputs/dNumericOutput_82
//     PlcTask Outputs/GVL.NumericOutput[83] <-> Outputs/dNumericOutput_83
//     PlcTask Outputs/GVL.NumericOutput[84] <-> Outputs/dNumericOutput_84
//     PlcTask Outputs/GVL.NumericOutput[85] <-> Outputs/dNumericOutput_85
//     PlcTask Outputs/GVL.NumericOutput[86] <-> Outputs/dNumericOutput_86
//     PlcTask Outputs/GVL.NumericOutput[87] <-> Outputs/dNumericOutput_87
//     PlcTask Outputs/GVL.NumericOutput[88] <-> Outputs/dNumericOutput_88
//     PlcTask Outputs/GVL.NumericOutput[89] <-> Outputs/dNumericOutput_89
//     PlcTask Outputs/GVL.NumericOutput[8] <-> Outputs/dNumericOutput_8
//     PlcTask Outputs/GVL.NumericOutput[90] <-> Outputs/dNumericOutput_90
//     PlcTask Outputs/GVL.NumericOutput[91] <-> Outputs/dNumericOutput_91
//     PlcTask Outputs/GVL.NumericOutput[92] <-> Outputs/dNumericOutput_92
//     PlcTask Outputs/GVL.NumericOutput[93] <-> Outputs/dNumericOutput_93
//     PlcTask Outputs/GVL.NumericOutput[94] <-> Outputs/dNumericOutput_94
//     PlcTask Outputs/GVL.NumericOutput[95] <-> Outputs/dNumericOutput_95
//     PlcTask Outputs/GVL.NumericOutput[96] <-> Outputs/dNumericOutput_96
//     PlcTask Outputs/GVL.NumericOutput[97] <-> Outputs/dNumericOutput_97
//     PlcTask Outputs/GVL.NumericOutput[98] <-> Outputs/dNumericOutput_98
//     PlcTask Outputs/GVL.NumericOutput[99] <-> Outputs/dNumericOutput_99
//     PlcTask Outputs/GVL.NumericOutput[9] <-> Outputs/dNumericOutput_9
//     PlcTask Outputs/GVL.NumericOutput[{0..119}] @bit 16 <-> Outputs/iNumericOutput_{0..119}  (120 links)
//     PlcTask Outputs/GVL.NumericOutput[69] @bit 16 <-> Outputs/dNumericOutput_69
//   MorpheePanel_PowerSupplyControl/MorpheePanel_PowerSupplyControl Instance <-> Device 5 (EL6751)/DPU3200_ID3
//     PlcTask Inputs/GVL.Bus1_Devices_Rx[0]/Command <-> ResponseSixBytes_id3/Inputs/command_code
//     PlcTask Inputs/GVL.Bus1_Devices_Rx[0]/Data[0] <-> ResponseSixBytes_id3/Inputs/data_6bytes
//     PlcTask Inputs/GVL.Bus1_Devices_Rx[0]/Data[{1..5}] <-> ResponseSixBytes_id3/Inputs/data_6bytes @bit {8..40 step 8}  (5 links)
//     PlcTask Outputs/GVL.Bus1_Devices[0]/Command <-> CommandNoDataBytes_id3/Outputs/command_code
//     PlcTask Outputs/GVL.Bus1_Devices_DLC3[0]/Command <-> CommandOneDataByte_id3/Outputs/command_code
//     PlcTask Outputs/GVL.Bus1_Devices_DLC3[0]/Data[0] <-> CommandOneDataByte_id3/Outputs/data_single
//     PlcTask Outputs/GVL.Bus1_Devices_DLC4[0]/Command <-> CommandTwoDataBytes_id3/Outputs/command_code
//     PlcTask Outputs/GVL.Bus1_Devices_DLC4[0]/Data[0] <-> CommandTwoDataBytes_id3/Outputs/data_word
//     PlcTask Outputs/GVL.Bus1_Devices_DLC4[0]/Data[1] <-> CommandTwoDataBytes_id3/Outputs/data_word @bit 8
//   MorpheePanel_PowerSupplyControl/MorpheePanel_PowerSupplyControl Instance <-> Device 5 (EL6751)/DPU3200_ID5
//     PlcTask Inputs/GVL.Bus1_Devices_Rx[1]/Command <-> ResponseSixBytes_id5/Inputs/command_code
//     PlcTask Inputs/GVL.Bus1_Devices_Rx[1]/Data[0] <-> ResponseSixBytes_id5/Inputs/data_6bytes
//     PlcTask Inputs/GVL.Bus1_Devices_Rx[1]/Data[{1..5}] <-> ResponseSixBytes_id5/Inputs/data_6bytes @bit {8..40 step 8}  (5 links)
//     PlcTask Outputs/GVL.Bus1_Devices[1]/Command <-> CommandNoDataBytes_id5/Outputs/command_code
//     PlcTask Outputs/GVL.Bus1_Devices_DLC3[1]/Command <-> CommandOneDataByte_id5/Outputs/command_code
//     PlcTask Outputs/GVL.Bus1_Devices_DLC3[1]/Data[0] <-> CommandOneDataByte_id5/Outputs/data_single
//     PlcTask Outputs/GVL.Bus1_Devices_DLC4[1]/Command <-> CommandTwoDataBytes_id5/Outputs/command_code
//     PlcTask Outputs/GVL.Bus1_Devices_DLC4[1]/Data[0] <-> CommandTwoDataBytes_id5/Outputs/data_word
//     PlcTask Outputs/GVL.Bus1_Devices_DLC4[1]/Data[1] <-> CommandTwoDataBytes_id5/Outputs/data_word @bit 8
//   MorpheePanel_PowerSupplyControl/MorpheePanel_PowerSupplyControl Instance <-> Device 5 (EL6751)/DPU3200_ID6
//     PlcTask Inputs/GVL.Bus1_Devices_Rx[2]/Command <-> ResponseSixBytes_id6/Inputs/command_code
//     PlcTask Inputs/GVL.Bus1_Devices_Rx[2]/Data[0] <-> ResponseSixBytes_id6/Inputs/data_6bytes
//     PlcTask Inputs/GVL.Bus1_Devices_Rx[2]/Data[{1..5}] <-> ResponseSixBytes_id6/Inputs/data_6bytes @bit {8..40 step 8}  (5 links)
//     PlcTask Outputs/GVL.Bus1_Devices[2]/Command <-> CommandNoDataBytes_id6/Outputs/command_code
//     PlcTask Outputs/GVL.Bus1_Devices_DLC3[2]/Command <-> CommandOneDataByte_id6/Outputs/command_code
//     PlcTask Outputs/GVL.Bus1_Devices_DLC3[2]/Data[0] <-> CommandOneDataByte_id6/Outputs/data_single
//     PlcTask Outputs/GVL.Bus1_Devices_DLC4[2]/Command <-> CommandTwoDataBytes_id6/Outputs/command_code
//     PlcTask Outputs/GVL.Bus1_Devices_DLC4[2]/Data[0] <-> CommandTwoDataBytes_id6/Outputs/data_word
//     PlcTask Outputs/GVL.Bus1_Devices_DLC4[2]/Data[1] <-> CommandTwoDataBytes_id6/Outputs/data_word @bit 8
//   MorpheePanel_PowerSupplyControl/MorpheePanel_PowerSupplyControl Instance <-> Device 5 (EL6751)/DPU3200_ID7
//     PlcTask Inputs/GVL.Bus1_Devices_Rx[3]/Command <-> ResponseSixBytes_id7/Inputs/command_code
//     PlcTask Inputs/GVL.Bus1_Devices_Rx[3]/Data[0] <-> ResponseSixBytes_id7/Inputs/data_6bytes
//     PlcTask Inputs/GVL.Bus1_Devices_Rx[3]/Data[{1..5}] <-> ResponseSixBytes_id7/Inputs/data_6bytes @bit {8..40 step 8}  (5 links)
//     PlcTask Outputs/GVL.Bus1_Devices[3]/Command <-> CommandNoDataBytes_id7/Outputs/command_code
//     PlcTask Outputs/GVL.Bus1_Devices_DLC3[3]/Command <-> CommandOneDataByte_id7/Outputs/command_code
//     PlcTask Outputs/GVL.Bus1_Devices_DLC3[3]/Data[0] <-> CommandOneDataByte_id7/Outputs/data_single
//     PlcTask Outputs/GVL.Bus1_Devices_DLC4[3]/Command <-> CommandTwoDataBytes_id7/Outputs/command_code
//     PlcTask Outputs/GVL.Bus1_Devices_DLC4[3]/Data[0] <-> CommandTwoDataBytes_id7/Outputs/data_word
//     PlcTask Outputs/GVL.Bus1_Devices_DLC4[3]/Data[1] <-> CommandTwoDataBytes_id7/Outputs/data_word @bit 8
//   MorpheePanel_PowerSupplyControl/MorpheePanel_PowerSupplyControl Instance <-> Device 6 (EL6751)/BIC2200_ID0
//     PlcTask Inputs/GVL.Bus2_Devices_Rx[0]/Command <-> ResponseSixBytes_id0/Inputs/command_code
//     PlcTask Inputs/GVL.Bus2_Devices_Rx[0]/Data[0] <-> ResponseSixBytes_id0/Inputs/data_6bytes
//     PlcTask Inputs/GVL.Bus2_Devices_Rx[0]/Data[{1..5}] <-> ResponseSixBytes_id0/Inputs/data_6bytes @bit {8..40 step 8}  (5 links)
//     PlcTask Outputs/GVL.Bus2_Devices[0]/Command <-> CommandNoDataBytes_id0/Outputs/command_code
//     PlcTask Outputs/GVL.Bus2_Devices_DLC3[0]/Command <-> CommandOneDataByte_id0/Outputs/command_code
//     PlcTask Outputs/GVL.Bus2_Devices_DLC3[0]/Data[0] <-> CommandOneDataByte_id0/Outputs/data_single
//     PlcTask Outputs/GVL.Bus2_Devices_DLC4[0]/Command <-> CommandTwoDataBytes_id0/Outputs/command_code
//     PlcTask Outputs/GVL.Bus2_Devices_DLC4[0]/Data[0] <-> CommandTwoDataBytes_id0/Outputs/data_word
//     PlcTask Outputs/GVL.Bus2_Devices_DLC4[0]/Data[1] <-> CommandTwoDataBytes_id0/Outputs/data_word @bit 8
//   MorpheePanel_PowerSupplyControl/MorpheePanel_PowerSupplyControl Instance <-> Device 6 (EL6751)/BIC2200_ID1
//     PlcTask Inputs/GVL.Bus2_Devices_Rx[1]/Command <-> ResponseSixBytes_id1/Inputs/command_code
//     PlcTask Inputs/GVL.Bus2_Devices_Rx[1]/Data[0] <-> ResponseSixBytes_id1/Inputs/data_6bytes
//     PlcTask Inputs/GVL.Bus2_Devices_Rx[1]/Data[{1..5}] <-> ResponseSixBytes_id1/Inputs/data_6bytes @bit {8..40 step 8}  (5 links)
//     PlcTask Outputs/GVL.Bus2_Devices[1]/Command <-> CommandNoDataBytes_id1/Outputs/command_code
//     PlcTask Outputs/GVL.Bus2_Devices_DLC3[1]/Command <-> CommandOneDataByte_id1/Outputs/command_code
//     PlcTask Outputs/GVL.Bus2_Devices_DLC3[1]/Data[0] <-> CommandOneDataByte_id1/Outputs/data_single
//     PlcTask Outputs/GVL.Bus2_Devices_DLC4[1]/Command <-> CommandTwoDataBytes_id1/Outputs/command_code
//     PlcTask Outputs/GVL.Bus2_Devices_DLC4[1]/Data[0] <-> CommandTwoDataBytes_id1/Outputs/data_word
//     PlcTask Outputs/GVL.Bus2_Devices_DLC4[1]/Data[1] <-> CommandTwoDataBytes_id1/Outputs/data_word @bit 8
//   MorpheePanel_PowerSupplyControl/MorpheePanel_PowerSupplyControl Instance <-> Device 6 (EL6751)/BIC2200_ID2
//     PlcTask Inputs/GVL.Bus2_Devices_Rx[2]/Command <-> ResponseSixBytes_id2/Inputs/command_code
//     PlcTask Inputs/GVL.Bus2_Devices_Rx[2]/Data[0] <-> ResponseSixBytes_id2/Inputs/data_6bytes
//     PlcTask Inputs/GVL.Bus2_Devices_Rx[2]/Data[{1..5}] <-> ResponseSixBytes_id2/Inputs/data_6bytes @bit {8..40 step 8}  (5 links)
//     PlcTask Outputs/GVL.Bus2_Devices[2]/Command <-> CommandNoDataBytes_id2/Outputs/command_code
//     PlcTask Outputs/GVL.Bus2_Devices_DLC3[2]/Command <-> CommandOneDataByte_id2/Outputs/command_code
//     PlcTask Outputs/GVL.Bus2_Devices_DLC3[2]/Data[0] <-> CommandOneDataByte_id2/Outputs/data_single
//     PlcTask Outputs/GVL.Bus2_Devices_DLC4[2]/Command <-> CommandTwoDataBytes_id2/Outputs/command_code
//     PlcTask Outputs/GVL.Bus2_Devices_DLC4[2]/Data[0] <-> CommandTwoDataBytes_id2/Outputs/data_word
//     PlcTask Outputs/GVL.Bus2_Devices_DLC4[2]/Data[1] <-> CommandTwoDataBytes_id2/Outputs/data_word @bit 8
//   MorpheePanel_PowerSupplyControl/MorpheePanel_PowerSupplyControl Instance <-> Device 6 (EL6751)/BIC2200_ID3
//     PlcTask Inputs/GVL.Bus2_Devices_Rx[3]/Command <-> ResponseSixBytes_id3/Inputs/command_code
//     PlcTask Inputs/GVL.Bus2_Devices_Rx[3]/Data[0] <-> ResponseSixBytes_id3/Inputs/data_6bytes
//     PlcTask Inputs/GVL.Bus2_Devices_Rx[3]/Data[{1..5}] <-> ResponseSixBytes_id3/Inputs/data_6bytes @bit {8..40 step 8}  (5 links)
//     PlcTask Outputs/GVL.Bus2_Devices[3]/Command <-> CommandNoDataBytes_id3/Outputs/command_code
//     PlcTask Outputs/GVL.Bus2_Devices_DLC3[3]/Command <-> CommandOneDataByte_id3/Outputs/command_code
//     PlcTask Outputs/GVL.Bus2_Devices_DLC3[3]/Data[0] <-> CommandOneDataByte_id3/Outputs/data_single
//     PlcTask Outputs/GVL.Bus2_Devices_DLC4[3]/Command <-> CommandTwoDataBytes_id3/Outputs/command_code
//     PlcTask Outputs/GVL.Bus2_Devices_DLC4[3]/Data[0] <-> CommandTwoDataBytes_id3/Outputs/data_word
//     PlcTask Outputs/GVL.Bus2_Devices_DLC4[3]/Data[1] <-> CommandTwoDataBytes_id3/Outputs/data_word @bit 8
//   MorpheePanel_PowerSupplyControl/MorpheePanel_PowerSupplyControl Instance <-> Device 6 (EL6751)/BIC2200_ID4
//     PlcTask Inputs/GVL.Bus2_Devices_Rx[4]/Command <-> ResponseSixBytes_id4/Inputs/command_code
//     PlcTask Inputs/GVL.Bus2_Devices_Rx[4]/Data[0] <-> ResponseSixBytes_id4/Inputs/data_6bytes
//     PlcTask Inputs/GVL.Bus2_Devices_Rx[4]/Data[{1..5}] <-> ResponseSixBytes_id4/Inputs/data_6bytes @bit {8..40 step 8}  (5 links)
//     PlcTask Outputs/GVL.Bus2_Devices[4]/Command <-> CommandNoDataBytes_id4/Outputs/command_code
//     PlcTask Outputs/GVL.Bus2_Devices_DLC3[4]/Command <-> CommandOneDataByte_id4/Outputs/command_code
//     PlcTask Outputs/GVL.Bus2_Devices_DLC3[4]/Data[0] <-> CommandOneDataByte_id4/Outputs/data_single
//     PlcTask Outputs/GVL.Bus2_Devices_DLC4[4]/Command <-> CommandTwoDataBytes_id4/Outputs/command_code
//     PlcTask Outputs/GVL.Bus2_Devices_DLC4[4]/Data[0] <-> CommandTwoDataBytes_id4/Outputs/data_word
//     PlcTask Outputs/GVL.Bus2_Devices_DLC4[4]/Data[1] <-> CommandTwoDataBytes_id4/Outputs/data_word @bit 8
//   MorpheePanel_PowerSupplyControl/MorpheePanel_PowerSupplyControl Instance <-> Device 6 (EL6751)/BIC2200_ID5
//     PlcTask Inputs/GVL.Bus2_Devices_Rx[5]/Command <-> ResponseSixBytes_id5/Inputs/command_code
//     PlcTask Inputs/GVL.Bus2_Devices_Rx[5]/Data[0] <-> ResponseSixBytes_id5/Inputs/data_6bytes
//     PlcTask Inputs/GVL.Bus2_Devices_Rx[5]/Data[{1..5}] <-> ResponseSixBytes_id5/Inputs/data_6bytes @bit {8..40 step 8}  (5 links)
//     PlcTask Outputs/GVL.Bus2_Devices[5]/Command <-> CommandNoDataBytes_id5/Outputs/command_code
//     PlcTask Outputs/GVL.Bus2_Devices_DLC3[5]/Command <-> CommandOneDataByte_id5/Outputs/command_code
//     PlcTask Outputs/GVL.Bus2_Devices_DLC3[5]/Data[0] <-> CommandOneDataByte_id5/Outputs/data_single
//     PlcTask Outputs/GVL.Bus2_Devices_DLC4[5]/Command <-> CommandTwoDataBytes_id5/Outputs/command_code
//     PlcTask Outputs/GVL.Bus2_Devices_DLC4[5]/Data[0] <-> CommandTwoDataBytes_id5/Outputs/data_word
//     PlcTask Outputs/GVL.Bus2_Devices_DLC4[5]/Data[1] <-> CommandTwoDataBytes_id5/Outputs/data_word @bit 8
//   MorpheePanel_PowerSupplyControl/MorpheePanel_PowerSupplyControl Instance <-> Device 6 (EL6751)/BIC2200_ID6
//     PlcTask Inputs/GVL.Bus2_Devices_Rx[6]/Command <-> ResponseSixBytes_id6/Inputs/command_code
//     PlcTask Inputs/GVL.Bus2_Devices_Rx[6]/Data[0] <-> ResponseSixBytes_id6/Inputs/data_6bytes
//     PlcTask Inputs/GVL.Bus2_Devices_Rx[6]/Data[{1..5}] <-> ResponseSixBytes_id6/Inputs/data_6bytes @bit {8..40 step 8}  (5 links)
//     PlcTask Outputs/GVL.Bus2_Devices[6]/Command <-> CommandNoDataBytes_id6/Outputs/command_code
//     PlcTask Outputs/GVL.Bus2_Devices_DLC3[6]/Command <-> CommandOneDataByte_id6/Outputs/command_code
//     PlcTask Outputs/GVL.Bus2_Devices_DLC3[6]/Data[0] <-> CommandOneDataByte_id6/Outputs/data_single
//     PlcTask Outputs/GVL.Bus2_Devices_DLC4[6]/Command <-> CommandTwoDataBytes_id6/Outputs/command_code
//     PlcTask Outputs/GVL.Bus2_Devices_DLC4[6]/Data[0] <-> CommandTwoDataBytes_id6/Outputs/data_word
//     PlcTask Outputs/GVL.Bus2_Devices_DLC4[6]/Data[1] <-> CommandTwoDataBytes_id6/Outputs/data_word @bit 8
//   MorpheePanel_PowerSupplyControl/MorpheePanel_PowerSupplyControl Instance <-> Device 6 (EL6751)/BIC2200_ID7
//     PlcTask Inputs/GVL.Bus2_Devices_Rx[7]/Command <-> ResponseSixBytes_id7/Inputs/command_code
//     PlcTask Inputs/GVL.Bus2_Devices_Rx[7]/Data[0] <-> ResponseSixBytes_id7/Inputs/data_6bytes
//     PlcTask Inputs/GVL.Bus2_Devices_Rx[7]/Data[{1..5}] <-> ResponseSixBytes_id7/Inputs/data_6bytes @bit {8..40 step 8}  (5 links)
//     PlcTask Outputs/GVL.Bus2_Devices[7]/Command <-> CommandNoDataBytes_id7/Outputs/command_code
//     PlcTask Outputs/GVL.Bus2_Devices_DLC3[7]/Command <-> CommandOneDataByte_id7/Outputs/command_code
//     PlcTask Outputs/GVL.Bus2_Devices_DLC3[7]/Data[0] <-> CommandOneDataByte_id7/Outputs/data_single
//     PlcTask Outputs/GVL.Bus2_Devices_DLC4[7]/Command <-> CommandTwoDataBytes_id7/Outputs/command_code
//     PlcTask Outputs/GVL.Bus2_Devices_DLC4[7]/Data[0] <-> CommandTwoDataBytes_id7/Outputs/data_word
//     PlcTask Outputs/GVL.Bus2_Devices_DLC4[7]/Data[1] <-> CommandTwoDataBytes_id7/Outputs/data_word @bit 8
//   MorpheePanel_PowerSupplyControl/MorpheePanel_PowerSupplyControl Instance <-> Device 7 (EL6751)/BIC2200_ID0
//     PlcTask Inputs/GVL.Bus3_Devices_Rx[0]/Command <-> ResponseSixBytes_id0/Inputs/command_code
//     PlcTask Inputs/GVL.Bus3_Devices_Rx[0]/Data[0] <-> ResponseSixBytes_id0/Inputs/data_6bytes
//     PlcTask Inputs/GVL.Bus3_Devices_Rx[0]/Data[{1..5}] <-> ResponseSixBytes_id0/Inputs/data_6bytes @bit {8..40 step 8}  (5 links)
//     PlcTask Outputs/GVL.Bus3_Devices[0]/Command <-> CommandNoDataBytes_id0/Outputs/command_code
//     PlcTask Outputs/GVL.Bus3_Devices_DLC3[0]/Command <-> CommandOneDataByte_id0/Outputs/command_code
//     PlcTask Outputs/GVL.Bus3_Devices_DLC3[0]/Data[0] <-> CommandOneDataByte_id0/Outputs/data_single
//     PlcTask Outputs/GVL.Bus3_Devices_DLC4[0]/Command <-> CommandTwoDataBytes_id0/Outputs/command_code
//     PlcTask Outputs/GVL.Bus3_Devices_DLC4[0]/Data[0] <-> CommandTwoDataBytes_id0/Outputs/data_word
//     PlcTask Outputs/GVL.Bus3_Devices_DLC4[0]/Data[1] <-> CommandTwoDataBytes_id0/Outputs/data_word @bit 8
//   MorpheePanel_PowerSupplyControl/MorpheePanel_PowerSupplyControl Instance <-> Device 7 (EL6751)/BIC2200_ID1
//     PlcTask Inputs/GVL.Bus3_Devices_Rx[1]/Command <-> ResponseSixBytes_id1/Inputs/command_code
//     PlcTask Inputs/GVL.Bus3_Devices_Rx[1]/Data[0] <-> ResponseSixBytes_id1/Inputs/data_6bytes
//     PlcTask Inputs/GVL.Bus3_Devices_Rx[1]/Data[{1..5}] <-> ResponseSixBytes_id1/Inputs/data_6bytes @bit {8..40 step 8}  (5 links)
//     PlcTask Outputs/GVL.Bus3_Devices[1]/Command <-> CommandNoDataBytes_id1/Outputs/command_code
//     PlcTask Outputs/GVL.Bus3_Devices_DLC3[1]/Command <-> CommandOneDataByte_id1/Outputs/command_code
//     PlcTask Outputs/GVL.Bus3_Devices_DLC3[1]/Data[0] <-> CommandOneDataByte_id1/Outputs/data_single
//     PlcTask Outputs/GVL.Bus3_Devices_DLC4[1]/Command <-> CommandTwoDataBytes_id1/Outputs/command_code
//     PlcTask Outputs/GVL.Bus3_Devices_DLC4[1]/Data[0] <-> CommandTwoDataBytes_id1/Outputs/data_word
//     PlcTask Outputs/GVL.Bus3_Devices_DLC4[1]/Data[1] <-> CommandTwoDataBytes_id1/Outputs/data_word @bit 8
//   MorpheePanel_PowerSupplyControl/MorpheePanel_PowerSupplyControl Instance <-> Device 7 (EL6751)/BIC2200_ID2
//     PlcTask Inputs/GVL.Bus3_Devices_Rx[2]/Command <-> ResponseSixBytes_id2/Inputs/command_code
//     PlcTask Inputs/GVL.Bus3_Devices_Rx[2]/Data[0] <-> ResponseSixBytes_id2/Inputs/data_6bytes
//     PlcTask Inputs/GVL.Bus3_Devices_Rx[2]/Data[{1..5}] <-> ResponseSixBytes_id2/Inputs/data_6bytes @bit {8..40 step 8}  (5 links)
//     PlcTask Outputs/GVL.Bus3_Devices[2]/Command <-> CommandNoDataBytes_id2/Outputs/command_code
//     PlcTask Outputs/GVL.Bus3_Devices_DLC3[2]/Command <-> CommandOneDataByte_id2/Outputs/command_code
//     PlcTask Outputs/GVL.Bus3_Devices_DLC3[2]/Data[0] <-> CommandOneDataByte_id2/Outputs/data_single
//     PlcTask Outputs/GVL.Bus3_Devices_DLC4[2]/Command <-> CommandTwoDataBytes_id2/Outputs/command_code
//     PlcTask Outputs/GVL.Bus3_Devices_DLC4[2]/Data[0] <-> CommandTwoDataBytes_id2/Outputs/data_word
//     PlcTask Outputs/GVL.Bus3_Devices_DLC4[2]/Data[1] <-> CommandTwoDataBytes_id2/Outputs/data_word @bit 8
//   MorpheePanel_PowerSupplyControl/MorpheePanel_PowerSupplyControl Instance <-> Device 7 (EL6751)/BIC2200_ID3
//     PlcTask Inputs/GVL.Bus3_Devices_Rx[3]/Command <-> ResponseSixBytes_id3/Inputs/command_code
//     PlcTask Inputs/GVL.Bus3_Devices_Rx[3]/Data[0] <-> ResponseSixBytes_id3/Inputs/data_6bytes
//     PlcTask Inputs/GVL.Bus3_Devices_Rx[3]/Data[{1..5}] <-> ResponseSixBytes_id3/Inputs/data_6bytes @bit {8..40 step 8}  (5 links)
//     PlcTask Outputs/GVL.Bus3_Devices[3]/Command <-> CommandNoDataBytes_id3/Outputs/command_code
//     PlcTask Outputs/GVL.Bus3_Devices_DLC3[3]/Command <-> CommandOneDataByte_id3/Outputs/command_code
//     PlcTask Outputs/GVL.Bus3_Devices_DLC3[3]/Data[0] <-> CommandOneDataByte_id3/Outputs/data_single
//     PlcTask Outputs/GVL.Bus3_Devices_DLC4[3]/Command <-> CommandTwoDataBytes_id3/Outputs/command_code
//     PlcTask Outputs/GVL.Bus3_Devices_DLC4[3]/Data[0] <-> CommandTwoDataBytes_id3/Outputs/data_word
//     PlcTask Outputs/GVL.Bus3_Devices_DLC4[3]/Data[1] <-> CommandTwoDataBytes_id3/Outputs/data_word @bit 8
//   MorpheePanel_PowerSupplyControl/MorpheePanel_PowerSupplyControl Instance <-> Device 7 (EL6751)/BIC2200_ID4
//     PlcTask Inputs/GVL.Bus3_Devices_Rx[4]/Command <-> ResponseSixBytes_id4/Inputs/command_code
//     PlcTask Inputs/GVL.Bus3_Devices_Rx[4]/Data[0] <-> ResponseSixBytes_id4/Inputs/data_6bytes
//     PlcTask Inputs/GVL.Bus3_Devices_Rx[4]/Data[{1..5}] <-> ResponseSixBytes_id4/Inputs/data_6bytes @bit {8..40 step 8}  (5 links)
//     PlcTask Outputs/GVL.Bus3_Devices[4]/Command <-> CommandNoDataBytes_id4/Outputs/command_code
//     PlcTask Outputs/GVL.Bus3_Devices_DLC3[4]/Command <-> CommandOneDataByte_id4/Outputs/command_code
//     PlcTask Outputs/GVL.Bus3_Devices_DLC3[4]/Data[0] <-> CommandOneDataByte_id4/Outputs/data_single
//     PlcTask Outputs/GVL.Bus3_Devices_DLC4[4]/Command <-> CommandTwoDataBytes_id4/Outputs/command_code
//     PlcTask Outputs/GVL.Bus3_Devices_DLC4[4]/Data[0] <-> CommandTwoDataBytes_id4/Outputs/data_word
//     PlcTask Outputs/GVL.Bus3_Devices_DLC4[4]/Data[1] <-> CommandTwoDataBytes_id4/Outputs/data_word @bit 8
//   MorpheePanel_PowerSupplyControl/MorpheePanel_PowerSupplyControl Instance <-> Device 7 (EL6751)/BIC2200_ID5
//     PlcTask Inputs/GVL.Bus3_Devices_Rx[5]/Command <-> ResponseSixBytes_id5/Inputs/command_code
//     PlcTask Inputs/GVL.Bus3_Devices_Rx[5]/Data[0] <-> ResponseSixBytes_id5/Inputs/data_6bytes
//     PlcTask Inputs/GVL.Bus3_Devices_Rx[5]/Data[{1..5}] <-> ResponseSixBytes_id5/Inputs/data_6bytes @bit {8..40 step 8}  (5 links)
//     PlcTask Outputs/GVL.Bus3_Devices[5]/Command <-> CommandNoDataBytes_id5/Outputs/command_code
//     PlcTask Outputs/GVL.Bus3_Devices_DLC3[5]/Command <-> CommandOneDataByte_id5/Outputs/command_code
//     PlcTask Outputs/GVL.Bus3_Devices_DLC3[5]/Data[0] <-> CommandOneDataByte_id5/Outputs/data_single
//     PlcTask Outputs/GVL.Bus3_Devices_DLC4[5]/Command <-> CommandTwoDataBytes_id5/Outputs/command_code
//     PlcTask Outputs/GVL.Bus3_Devices_DLC4[5]/Data[0] <-> CommandTwoDataBytes_id5/Outputs/data_word
//     PlcTask Outputs/GVL.Bus3_Devices_DLC4[5]/Data[1] <-> CommandTwoDataBytes_id5/Outputs/data_word @bit 8
//   MorpheePanel_PowerSupplyControl/MorpheePanel_PowerSupplyControl Instance <-> Device 7 (EL6751)/BIC2200_ID6
//     PlcTask Inputs/GVL.Bus3_Devices_Rx[6]/Command <-> ResponseSixBytes_id6/Inputs/command_code
//     PlcTask Inputs/GVL.Bus3_Devices_Rx[6]/Data[0] <-> ResponseSixBytes_id6/Inputs/data_6bytes
//     PlcTask Inputs/GVL.Bus3_Devices_Rx[6]/Data[{1..5}] <-> ResponseSixBytes_id6/Inputs/data_6bytes @bit {8..40 step 8}  (5 links)
//     PlcTask Outputs/GVL.Bus3_Devices[6]/Command <-> CommandNoDataBytes_id6/Outputs/command_code
//     PlcTask Outputs/GVL.Bus3_Devices_DLC3[6]/Command <-> CommandOneDataByte_id6/Outputs/command_code
//     PlcTask Outputs/GVL.Bus3_Devices_DLC3[6]/Data[0] <-> CommandOneDataByte_id6/Outputs/data_single
//     PlcTask Outputs/GVL.Bus3_Devices_DLC4[6]/Command <-> CommandTwoDataBytes_id6/Outputs/command_code
//     PlcTask Outputs/GVL.Bus3_Devices_DLC4[6]/Data[0] <-> CommandTwoDataBytes_id6/Outputs/data_word
//     PlcTask Outputs/GVL.Bus3_Devices_DLC4[6]/Data[1] <-> CommandTwoDataBytes_id6/Outputs/data_word @bit 8
//   MorpheePanel_PowerSupplyControl/MorpheePanel_PowerSupplyControl Instance <-> Device 7 (EL6751)/BIC2200_ID7
//     PlcTask Inputs/GVL.Bus3_Devices_Rx[7]/Command <-> ResponseSixBytes_id7/Inputs/command_code
//     PlcTask Inputs/GVL.Bus3_Devices_Rx[7]/Data[0] <-> ResponseSixBytes_id7/Inputs/data_6bytes
//     PlcTask Inputs/GVL.Bus3_Devices_Rx[7]/Data[{1..5}] <-> ResponseSixBytes_id7/Inputs/data_6bytes @bit {8..40 step 8}  (5 links)
//     PlcTask Outputs/GVL.Bus3_Devices[7]/Command <-> CommandNoDataBytes_id7/Outputs/command_code
//     PlcTask Outputs/GVL.Bus3_Devices_DLC3[7]/Command <-> CommandOneDataByte_id7/Outputs/command_code
//     PlcTask Outputs/GVL.Bus3_Devices_DLC3[7]/Data[0] <-> CommandOneDataByte_id7/Outputs/data_single
//     PlcTask Outputs/GVL.Bus3_Devices_DLC4[7]/Command <-> CommandTwoDataBytes_id7/Outputs/command_code
//     PlcTask Outputs/GVL.Bus3_Devices_DLC4[7]/Data[0] <-> CommandTwoDataBytes_id7/Outputs/data_word
//     PlcTask Outputs/GVL.Bus3_Devices_DLC4[7]/Data[1] <-> CommandTwoDataBytes_id7/Outputs/data_word @bit 8

CONFIGURATION MorpheePanel_PowerSupplyControl
    RESOURCE PLC ON TwinCAT3
        TASK PlcTask(INTERVAL := T#10ms, PRIORITY := 20);
        PROGRAM Main WITH PlcTask : Main;
    END_RESOURCE
END_CONFIGURATION

// ---- DUTs/panel302.TcDUT
TYPE panel302 :
STRUCT
	rxdata : ARRAY[0..101] OF UINT;
	txdata : ARRAY[0..89] OF UINT;
END_STRUCT
END_TYPE

// ---- DUTs/RxData.TcDUT
TYPE RxData :
STRUCT
  Command : UINT;         // Echoed command code
  Data : ARRAY[0..5] OF BYTE; // 6 bytes for response data
END_STRUCT
END_TYPE

// ---- DUTs/TxData.TcDUT
TYPE TxData :
STRUCT
  Command : INT;                     // Command index (2 bytes: )
  Data : ARRAY[0..3] OF BYTE;        // Data payload as 4 bytes (Command + Data + padding if needed)
END_STRUCT
END_TYPE

// ---- GVLs/GVL.TcGVL
VAR_GLOBAL
    AdlOn: ARRAY[0..19] OF BOOL;          (** Active dummy load control status: 0 = off/not supported, 1 = on **)
    AlarmStatus: UINT;                    (** Bitmask of active alarms, 1 bit per device **)
    Bus1_Devices AT %Q*: ARRAY[0..3] OF TxData; (** CAN Bus 1 Tx data for devices 0-3 **)
    Bus1_Devices_DLC3 AT %Q*: ARRAY[0..3] OF TxData; (** CAN Bus 1 DLC 3 commands **)
    Bus1_Devices_DLC4 AT %Q*: ARRAY[0..3] OF TxData; (** CAN Bus 1 DLC 4 commands **)
    Bus1_Devices_Rx AT %I*: ARRAY[0..3] OF RxData; (** CAN Bus 1 Rx data **)
    Bus2_Devices AT %Q*: ARRAY[0..7] OF TxData; (** CAN Bus 2 Tx data for devices 4-11 **)
    Bus2_Devices_DLC3 AT %Q*: ARRAY[0..7] OF TxData; (** CAN Bus 2 DLC 3 commands **)
    Bus2_Devices_DLC4 AT %Q*: ARRAY[0..7] OF TxData; (** CAN Bus 2 DLC 4 commands **)
    Bus2_Devices_Rx AT %I*: ARRAY[0..7] OF RxData; (** CAN Bus 2 Rx data **)
    Bus3_Devices AT %Q*: ARRAY[0..7] OF TxData; (** CAN Bus 3 Tx data for devices 12-19 **)
    Bus3_Devices_DLC3 AT %Q*: ARRAY[0..7] OF TxData; (** CAN Bus 3 DLC 3 commands **)
    Bus3_Devices_DLC4 AT %Q*: ARRAY[0..7] OF TxData; (** CAN Bus 3 DLC 4 commands **)
    Bus3_Devices_Rx AT %I*: ARRAY[0..7] OF RxData; (** CAN Bus 3 Rx data **)
    CommFault: ARRAY[0..19] OF BOOL;      (** Communication fault per device **)
    CommTimeouts: ARRAY[0..19] OF INT;    (** Communication timeouts per device **)
    Current: ARRAY[0..19] OF BOOL;        (** Device mode Current: 0 = not in Current mode, 1 = Current mode **)
    CurrentScale: ARRAY[0..19] OF UINT;
    DataValid: ARRAY[0..19] OF BOOL;      (** Data freshness status **)
    DcOk: ARRAY[0..19] OF BOOL;           (** Secondary DD output voltage status: 0 = TOO LOW, 1 = NORMAL **)
    DeviceFlags: ARRAY[0..19] OF BYTE;    (** Device status bits **)
    DeviceSystemFlags: ARRAY[0..19] OF UINT;(** Device status bits **)
    Direction: ARRAY[0..19] OF BOOL;      (** Direction control **)
    Eeper: ARRAY[0..19] OF BOOL;          (** EEPROM data access error: 0 = normal, 1 = error **)
 	 EL2809_InputFlags: ARRAY[0..2] OF WORD;     (** 3 16-bit flags for EL2809 channels **)
    EL2798_InputFlags: BYTE;              (** 8-bit flags for EL2798 channels **)
    EL2809_Output AT %Q*: ARRAY[0..3,0..15] OF BOOL;  (** 16-channel output for EL2809 **)
    EL2798_Output AT %Q*: ARRAY[0..7] OF BOOL;   (** 8-channel output for EL2798 **)
    EL3174_Channel1_Value AT %I* : INT;           (** Raw analog value from EL3174 channel 1, 0-10V **)
    EL3174_Channel2_Value: INT;           (** Raw analog value from EL3174 channel 2, 0-10V **)
    EL3174_Channel3_Value: INT;           (** Raw analog value from EL3174 channel 3, 0-10V **)
    EL3174_Channel4_Value: INT;           (** Raw analog value from EL3174 channel 4, 0-10V **)
    EL3174_Channel1_Alarm: BOOL;          (** Yellow alarm from GT, channel 1, >2.5V **)
    EL3174_Channel2_Alarm: BOOL;          (** Alarm for channel 2, >2.5V, optional **)
    EL3174_Channel3_Alarm: BOOL;          (** Alarm for channel 3, >2.5V, optional **)
    EL3174_Channel4_Alarm: BOOL;          (** Alarm for channel 4, >2.5V, optional **)
    EStop: ARRAY[0..19] OF BOOL;          (** Emergency stop per device **)
    EthercatAlive: BOOL;                  (** EtherCAT communication status **)
    EthercatAliveFromMaster: BOOL;        (** EtherCAT master status **)
    EthercatAslaveStatus AT %I*: UINT;    (** EtherCAT slave status **)
    FanSpeed1: ARRAY[0..19] OF UINT;      (** Fan 1 speed, RPM **)
    FanSpeed2: ARRAY[0..19] OF UINT;      (** Fan 2 speed, RPM **)
    FanSpeedScale: ARRAY[0..19] OF UINT;
    FaultLevel: ARRAY[0..19] OF BYTE;     (** Fault severity **)
    FaultStatus: ARRAY[0..19] OF UINT;    (** Fault status code **)
    FirstRun: BOOL := TRUE;               (** Initial PLC startup flag **)
    GroupCapacity: ARRAY[0..3] OF UINT;   (** CBU capacity, watts **)
    GroupCurrentLimit: ARRAY[0..3] OF UINT; (** CBU current limit, 0-270A **)
    GroupDemand: ARRAY[0..3] OF UINT;     (** CBU demand, watts **)
    GroupMaster: ARRAY[0..3] OF INT;      (** CBU master device index **)
    GroupVoltageLimit: ARRAY[0..3] OF UINT; (** CBU voltage limit, 24-32V **)
	IoutSetpoint: ARRAY[0..19] OF REAL;  
    Iin: ARRAY[0..19] OF UINT;
    IinScale: ARRAY[0..19] OF UINT;
    InitialState: ARRAY[0..19] OF BOOL;   (** Device initialized status: 0 = initializing, 1 = not initializing **)
    Iout: ARRAY[0..19] OF UINT;           (** Output current, raw **)
    GroupMembership: ARRAY[0..19] OF INT;
    IoutSetRev: ARRAY[0..19] OF REAL;     (** Reverse current setpoint, F=0.01 **)
    LastUpdateTime: ARRAY[0..19] OF TIME; (** Last valid data timestamp **)
    MfrSerialPersistent: ARRAY[0..19] OF ARRAY[0..53] OF BYTE; (** Persistent storage for manufacturer serial data **)
    Ms: ARRAY[0..19] OF BOOL;             (** Parallel mode status: 0 = Slave, 1 = Master **)
    MorpheeCANCommFault: BOOL;            (** Morphee CAN fault **)
    MorpheeCommFault: BOOL;               (** Morphee communication fault **)
    MorpheeDoorPGSArea: BOOL;             (** Morphee door PGS area **)
    MorpheeECUFault: BOOL;                (** Morphee ECU fault **)
    MorpheeElectricalFault: BOOL;         (** Morphee electrical fault **)
    MorpheeEStop: BOOL;                   (** Morphee E-Stop **)
    MorpheeFireAlarm: BOOL;               (** Morphee fire alarm **)
    MorpheeGasPGSAlarm: BOOL;             (** Morphee gas PGS alarm **)
    MorpheeMCUFault: BOOL;                (** Morphee MCU fault **)
    MorpheeScavengeFanFault: BOOL;        (** Morphee scavenge fan fault **)
    MorpheeWatchdogFault: BOOL;           (** Morphee watchdog fault **)
    NumericInput AT %I*: ARRAY[0..239] OF WORD; (** EtherCAT input data **)
    (* Temporary test inputs for groups: 4 groups x 7 inputs = 28 indices *)
    UseTempGroupInputs : BOOL := FALSE;        (** When TRUE, EthercatManager will read group inputs from TempGroupInput instead of NumericInput **)
    TempGroupInput : ARRAY[0..27] OF WORD;     (** Temporary group inputs mapping for testing; indexes 0..27 map to group base 10..37 **) 
    UseTempBus1Direct : BOOL := FALSE;         (** When TRUE, EthercatManager will read Bus1 device inputs from TempBus1* arrays instead of NumericInput **)
    TempBus1VoutSetpoint : ARRAY[0..3] OF WORD;(** Temporary Bus1 voltage setpoints, V*100 **)
    TempBus1IoutSetpoint : ARRAY[0..3] OF WORD;(** Temporary Bus1 current setpoints, A*100 **)
    TempBus1Flags : ARRAY[0..3] OF WORD;       (** Temporary Bus1 flags, same bit mapping as device flags **)
    TempBus1VoutSetMin : ARRAY[0..3] OF WORD;  (** Temporary Bus1 min voltage, V*100 **)
    TempBus1VoutSetMax : ARRAY[0..3] OF WORD;  (** Temporary Bus1 max voltage, V*100 **)
    TempBus1IoutSetMin : ARRAY[0..3] OF WORD;  (** Temporary Bus1 min current, A*100 **)
    TempBus1IoutSetMax : ARRAY[0..3] OF WORD;  (** Temporary Bus1 max current, A*100 **)
    NumericOutput AT %Q*: ARRAY[0..120] OF DWORD; (** EtherCAT output data **)
    OperationOn: ARRAY[0..19] OF BOOL;    (** Device operation status **)
    OrangeStop: ARRAY[0..19] OF BOOL;     (** Orange-level stop **)
    OutputOn: ARRAY[0..19] OF BOOL;       (** Output enabled status **)
    PfcOk: ARRAY[0..19] OF BOOL;          (** Primary PFC status: 0 = OFF/abnormal, 1 = ON normally **)
    PollingPaused: ARRAY[0..19] OF BOOL;  (** CAN polling pause **)
    PollingPauseTimeout: ARRAY[0..19] OF TON; (** Timeout for polling pause **)
    PollingPauseStartTime: ARRAY[0..19] OF TIME; (** Start time of polling pause **)
    ReadCommandIndex: ARRAY[0..19] OF INT; (** CAN read command index **)
    RecoveryPending: ARRAY[0..19] OF BOOL; (** Fault recovery pending **)
    RedStop: ARRAY[0..19] OF BOOL;        (** Red-level stop **)
    RemoteMasterAlive: BOOL;              (** Remote master status **)
    SafetyCANCommFault: BOOL;             (** Safety CAN fault **)
    SafetyDoorPGSArea: BOOL;              (** Safety door PGS area **)
    SafetyECUFault: BOOL;                 (** Safety ECU fault **)
    SafetyElectricalFault: BOOL;          (** Safety electrical fault **)
    SafetyEStop: INT;                     (** System E-Stop counter **)
    SafetyFireAlarm: BOOL;                (** Safety fire alarm **)
    SafetyGasPGSAlarm: BOOL;              (** Safety gas PGS alarm **)
    SafetyMCUFault: BOOL;                 (** Safety MCU fault **)
    SafetyOK: ARRAY[0..19] OF BOOL;       (** Device safe to operate **)
    SafetyRecovery: BOOL;                 (** Fault recovery status **)
    SafetyShutdown: ARRAY[0..19] OF BOOL; (** Device in safety shutdown **)
    Standby: ARRAY[0..19] OF BOOL;        (** Device mode Standby: 0 = not in Standby mode, 1 = Standby mode **)
    SuccessCounts: ARRAY[0..19] OF INT;   (** Successful polls per device **)
    SystemAlarms: UINT;                   (** System alarms bitfield **)
    SystemFlags: BYTE;                    (** System flags, bit 0 = maintenance **)
    SystemState: BYTE;                    (** System state: 0=normal, 1=orange, 2=red, 3=EStop **)
    TempScale: ARRAY[0..19] OF UINT;
    Temperature: ARRAY[0..19] OF UINT;    (** Device temperature, raw **)
    TemperatureFaultHigh AT %I*: ARRAY[0..19] OF BOOL; (** Hard-wired high temp fault **)
    Vin: ARRAY[0..19] OF UINT;            (** Input voltage, raw **)
    VinScale: ARRAY[0..19] OF UINT;
    Voltage: ARRAY[0..19] OF BOOL;        (** Device mode Voltage: 0 = not in Voltage mode, 1 = Voltage mode **)
    Vout: ARRAY[0..19] OF UINT;           (** Output voltage, raw **)
    VoutScale: ARRAY[0..19] OF UINT;
    VoutSetpoint: ARRAY[0..19] OF REAL;   (** Forward voltage setpoint, F=0.1 **)
    VoutSetRev: ARRAY[0..19] OF REAL;     (** Reverse voltage setpoint, F=0.01 **)
END_VAR

// ---- GVLs/GVL_Constant.TcGVL
VAR_GLOBAL CONSTANT
  CMD_BIDIRECTIONAL_CONFIG : UINT := 16#0140; (* R/W, 1 byte: Bidirectional config, DLC 3 *)
  CMD_DIRECTION_CTRL : UINT := 16#0100;     (* R/W, 1 byte: 00h=AC-to-DC, 01h=DC-to-AC, DLC 3 *)
  CMD_FAULT_STATUS : UINT := 16#0040;   (* R, 2 bytes: Fault status *)
  CMD_IOUT_SET : UINT := 16#0030;       (* R/W, 2 bytes: Current setpoint, DLC 4 *)
  CMD_MFR_DATE_B0B5 : UINT := 16#0086;      (* R/W, 6 bytes: Date *)
  CMD_MFR_ID_B0B5 : UINT := 16#0080;        (* R, 6 bytes: Manufacturer ID, bytes 0-5 *)
  CMD_MFR_ID_B6B11 : UINT := 16#0081;       (* R, 6 bytes: Manufacturer ID, bytes 6-11 *)
  CMD_MFR_LOCATION_B0B2 : UINT := 16#0085;  (* R/W, 3 bytes: Location *)
  CMD_MFR_MODEL_B0B5 : UINT := 16#0082;     (* R, 6 bytes: Model, bytes 0-5 *)
  CMD_MFR_MODEL_B6B11 : UINT := 16#0083;    (* R, 6 bytes: Model, bytes 6-11 *)
  CMD_MFR_REVISION_B0B5 : UINT := 16#0084;  (* R, 6 bytes: Revision, bytes 0-5 *)
  CMD_MFR_SERIAL_B0B5 : UINT := 16#0087;    (* R/W, 6 bytes: Serial number, bytes 0-5 *)
  CMD_MFR_SERIAL_B6B11 : UINT := 16#0088;   (* R/W, 6 bytes: Serial number, bytes 6-11 *)
  CMD_OPERATION : UINT := 16#0000;      (* R/W, 1 byte: 00h=OFF, 01h=ON, DLC 3 *)
  CMD_READ_FAN_SPEED1 : UINT := 16#0071;    (* R, 2 bytes: Fan 1 speed *)
  CMD_READ_FAN_SPEED2 : UINT := 16#0072;    (* R, 2 bytes: Fan 2 speed *)
  CMD_READ_IOUT : UINT := 16#0061;      (* R, 2 bytes: Output current, F=0.01 or 0.1 *)
  CMD_READ_TEMPERATURE_1 : UINT := 16#0062; (* R, 2 bytes: Temperature, F=0.1 *)
  CMD_READ_VIN : UINT := 16#0050;       (* R, 2 bytes: Input voltage, F=0.1 *)
  CMD_READ_VOUT : UINT := 16#0060;      (* R, 2 bytes: Output voltage, F=0.01 or 0.1 *)
  CMD_REVERSE_IOUT_SET : UINT := 16#0130;   (* R/W, 2 bytes: Reverse current setpoint, F=0.01, DLC 4 *)
  CMD_REVERSE_VOUT_SET : UINT := 16#0120;   (* R/W, 2 bytes: Reverse voltage setpoint, F=0.01, DLC 4 *)
  CMD_SCALING_FACTOR : UINT := 16#00C0;     (* R, 2 bytes: scaling factors (BIC models) *)
  CMD_SYSTEM_STATUS : UINT := 16#00C1;      (* R, 2 bytes: system status bits (M/S, DC_OK, PFC_OK, etc.) *)
  CMD_SYSTEM_CONFIG : UINT := 16#00C2;      (* R/W, 2 bytes: System configuration, DLC 4 *)
  CMD_VOUT_SET : UINT := 16#0020;       (* R/W, 2 bytes: Voltage setpoint, DLC 4 *)
  ESTOPTIME : TIME := T#10s;            (* Delay before E-Stop disables outputs *)
  HEARTBEATTIMEOUT : TIME := T#45ms;    (* Timeout for Morphee heartbeat *)
  IoutMax : UINT := 75;               (* Maximum current per BIC-2200 device, 2200A *)
  MAX_CURRENT : UINT := 270;            (* Maximum allowable current limit, 270A, unscaled, per CBU group *)
  MAX_VOLTAGE : UINT := 32;             (* Maximum allowable voltage limit, 32V, unscaled *)
  MAXCOMMSTALE : TIME := T#2s;          (* Threshold for stale communication data *)
  MAXCOMMTIMEOUT : UINT := 200;         (* Max comm timeouts before fault, 2s at 10ms cycle *)
  MfrCommands : ARRAY[0..8] OF UINT := [CMD_MFR_ID_B0B5, CMD_MFR_ID_B6B11, CMD_MFR_MODEL_B0B5,
                                        CMD_MFR_MODEL_B6B11, CMD_MFR_REVISION_B0B5, CMD_MFR_LOCATION_B0B2,
                                        CMD_MFR_DATE_B0B5, CMD_MFR_SERIAL_B0B5, CMD_MFR_SERIAL_B6B11]; (* Commands for Morphee initialization *)
  MIN_CURRENT : UINT := 0;              (* Minimum allowable current limit, 0A, unscaled *)
  MIN_VOLTAGE : UINT := 24;             (* Minimum allowable voltage limit, 24V, unscaled *)
  MINSUCCESSCLEAR : UINT := 3;          (* Minimum successful polls to clear fault *)
  MODE_CURRENT_FWD : BYTE := 1;         (* Current control, forward direction *)
  MODE_CURRENT_REV : BYTE := 3;         (* Current control, reverse direction *)
  MODE_STANDBY : BYTE := 0;             (* Standby mode *)
  MODE_VOLTAGE_FWD : BYTE := 2;         (* Voltage control, forward direction *)
  MODE_VOLTAGE_REV : BYTE := 4;         (* Voltage control, reverse direction *)
  OFFRAMP : TIME := T#10s;              (* Duration for OFF ramp-down *)
  ORANGESTOPTIME : TIME := T#3m;        (* Delay before Orange Stop disables outputs *)
  REDSTOPTIME : TIME := T#1m;           (* Delay before Red Stop disables outputs *)
  REMOTETIMEOUT : TIME := T#2s;         (* Timeout for RemoteMasterAlive *)
  SHUTDOWNRAMP : TIME := T#60s;         (* Duration for shutdown ramp-down *)
END_VAR

// ---- GVLs/GVL_Persistent.TcGVL
VAR_GLOBAL PERSISTENT
  MfrSerialInitDone : ARRAY[0..19] OF BOOL;                   // Flag indicating serial data initialization complete
  MfrSerialPersistent : ARRAY[0..19] OF ARRAY[0..53] OF BYTE; // Persistent storage for manufacturer serial data
  MfrSerialShared :BOOL;
  MfrSerialUpdated : BOOL;
END_VAR

// ---- GVLs/Safety_Tags.TcGVL
{attribute 'qualified_only'}
VAR_GLOBAL
	Reset AT %Q*: BOOL;
	Run AT %Q*: BOOL;
	
	Estop_ok AT %I*: BOOL;
	ECU1_2_Ok AT %I*: BOOL;
	CBU_LB_Ok AT %I*: BOOL;
	MCS_OK AT %I*: BOOL;
	
END_VAR

// ---- POU/Main.TcPOU

PROGRAM Main
VAR
  CycleCounter : INT := 0;                    // Counter for 100ms update cycle (10ms * 10)
  EthercatMgr : EthercatManager;              // EtherCAT manager instance
  SafetyMgr : SafetyMgr;                      // Safety manager instance
  GroupMgr : GroupManager;                    // Group manager instance
  Devices : ARRAY[0..19] OF DeviceManager;    // Array of device managers for CAN communication
  i : INT;                                    // Loop variable
END_VAR

Safety_Tags.Run := True;

IF  gvl.EthercatAslaveStatus>=4 THEN
	GVL.EthercatAlive:= TRUE;
ELSE
	GVL.EthercatAlive:= FALSE;
END_IF
// Initialize system on first run
IF GVL.FirstRun THEN
  FOR i := 0 TO 19 DO
    GVL.DeviceFlags[i] := 0;                  // Clear device flags
    IF i < 4 THEN
      GVL.Direction[i] := FALSE;              // Set initial direction: 0-3 AC-to-DC
    ELSE
      GVL.Direction[i] := TRUE;               // Set initial direction: 4-19 DC-to-AC
    END_IF;
   // GVL.DeviceMode[i] := GVL_Constant.MODE_STANDBY; // Start in standby mode
    Devices[i](DeviceIndex := i, Reset := TRUE);    // Initialize device manager with reset
    Devices[i].Poll();                        // Start polling CAN devices
  END_FOR;
  GVL.FirstRun := FALSE;                      // Mark initialization complete
END_IF;

// Main update loop (every 100ms)
CycleCounter := CycleCounter + 1;
IF CycleCounter >= 10 THEN
  FOR i := 0 TO 19 DO
    Devices[i](DeviceIndex := i, Reset := FALSE); // Update device managers without reset
    Devices[i].Poll();                        // Poll CAN devices for data
  END_FOR;
  SafetyMgr.UpdateSafety();                   // Update safety conditions
  GroupMgr.UpdateGroupMasters();              // Update group master assignments
  GroupMgr.UpdateGroupCapacity();             // Update group capacities and demands
  EthercatMgr.ProcessInputs();                // Process EtherCAT inputs
  EthercatMgr.UpdateOutputs();                // Update EtherCAT outputs
  // Commands are already sent inside EthercatMgr.ProcessInputs() via THIS^.ApplyCommands(...)
  SetpointTest();                             // TEMP: run setpoint test (remove when done)
  CycleCounter := 0;                          // Reset cycle counter
END_IF;

END_PROGRAM

// ---- POU/EthercatManager.TcPOU

FUNCTION_BLOCK EthercatManager
VAR
  IsInitPhase : BOOL := FALSE;               (* TRUE during initialization phase *)
  InitCycle : INT := 0;                      (* Current initialization cycle, 0-5 *)
  LastVoutSetpoint : ARRAY[0..19] OF UINT;   (* Last voltage setpoint sent *)
  LastIoutSetpoint : ARRAY[0..19] OF UINT;   (* Last current setpoint sent *)
  LastOutputOn : ARRAY[0..19] OF BOOL;       (* Last output enabled state *)
  LastOperationOn : ARRAY[0..19] OF BOOL;    (* Last operation state *)
  LastDirection : ARRAY[0..19] OF BOOL;      (* Last direction state *)
  fbDeviceManager : DeviceManager;           (* Device manager instance *)
  DataRefreshRequired : BOOL;                (* Flag for data refresh required *)
  RefreshTableRequired : BOOL;               (* Flag for table refresh required *)
  InitTimeout : TON;                         (* 10s timeout for init cycles *)
  LastMorpheeSignal : UINT;                  (* Track last Morphee signal *)
  VoutSetMin : ARRAY[0..19] OF UINT;		 (* Vout min limit *)
  VoutSetMax : ARRAY[0..19] OF UINT; 		 (* Vout max limit *)
  IoutSetMin : ARRAY[0..19] OF UINT; 		 (* Iout min limit *)
  IoutSetMax : ARRAY[0..19] OF UINT; 		 (* Iout max limit *)
  CanCtrlConfigured : ARRAY[0..19] OF BOOL; (* True after SYSTEM_CONFIG(0x00C2)=0x0003 is sent successfully *)
  commandData : UINT;                        (** Data to use for command **)
  LastCommandSentTime : ARRAY[0..19] OF TIME; (* Last successful write timestamp per device *)
END_VAR

(* Comment Section: GVL.NumericInput and GVL.NumericOutput Mapping *)
(* Purpose: This section provides a detailed reference for the GVL.NumericInput and GVL.NumericOutput *)
(* mappings used by the EthercatManager function block, including system inputs, group inputs, *)
(* device inputs, and output structures. All indices are carefully allocated to ensure no overlap *)
(* and to support the system's parallel configuration, maintenance mode, and group operation. *)

(* GVL.NumericInput Mapping *)
(* Overview: GVL.NumericInput stores system-wide inputs, group inputs, and device inputs for the *)
(* 20 power supply units (devices 0-19) and 4 groups (LVLA1-LVLA4). The allocation starts system *)
(* inputs at index 0, with group and device inputs starting at index 10. Each device and group *)
(* has 7 inputs to support setpoints, flags, and limits. *)

(* 0-4: System-Level Inputs and Reserves (5 indices) *)
(*   0: GVL.SystemAlarms (WORD to UINT) *)
(*      - Stores system-wide alarms, processed in ProcessInputs *)
(*   1: System Flags (WORD) *)
(*      - Bit 0 (16#0001): GVL.SystemFlags (includes maintenanceMode, set in ProcessInputs) *)
(*        - maintenanceMode = TRUE: Disables groups, uses individual device inputs *)
(*        - maintenanceMode = FALSE: Enables groups, master uses group inputs *)
(*      - Bit 1 (16#0002): GVL.EthercatAliveFromMaster (EtherCAT master status) *)
(*      - Bit 2 (16#0004): GVL.RemoteMasterAlive (Remote master status) *)
(*      - Bits 3-15: Unallocated (reserved for future flags) *)
(*   2: Morphee Initialization Signal (DWORD to UINT, processed in UpdateOutputs) *)
(*      - Values 1-5: Initialization cycle *)
(*      - Value 100: Complete initialization *)
(*   3-4: Reserved *)
(*      - Unallocated indices for future system-wide inputs *)
(* 5  EL2809 rack 1 slot 1
-9: Unallocated *)
(*      - Reserved for future system expansion *)
(* 10-37: Group Inputs (4 groups x 7 inputs = 28 indices) *)
(*   - Each group (LVLA1-LVLA4) has 7 inputs, treating the group as a single device in normal mode *)
(*   - For groupIdx = 0 TO 3, baseIdx = 10 + (groupIdx * 7): *)
(*     baseIdx: GroupVoutSetpoint (Voltage setpoint for group, applied to master) *)
(*     baseIdx + 1: GroupIoutSetpoint (Current setpoint for master, internally distributed) *)
(*     baseIdx + 2: Group Flags (WORD, similar to device flags) *)
(*       - Bit 0 (16#0001): GroupDirection (Forward/reverse, assumed) *)
(*       - Bit 1 (16#0002): GroupOperationOn (Operation active, assumed) *)
(*       - Bits 2-3 (16#000C): GroupDeviceMode (0-3, assumed) *)
(*       - Bit 7 (16#0080): GroupEStop (Assumed) *)
(*     baseIdx + 3: GroupVoutSetMin (Minimum voltage limit for master) *)
(*     baseIdx + 4: GroupVoutSetMax (Maximum voltage limit for master) *)
(*     baseIdx + 5: GroupIoutSetMin (Minimum current limit for master) *)
(*     baseIdx + 6: GroupIoutSetMax (Maximum current limit, constrained by GVL.GroupCapacity) *)
(*   - Group Index Breakdown: *)
(*     LVLA1 (groupIdx = 0): 10-16 *)
(*     LVLA2 (groupIdx = 1): 17-23 *)
(*     LVLA3 (groupIdx = 2): 24-30 *)
(*     LVLA4 (groupIdx = 3): 31-37 *)
(*   - Note: GroupIoutSetMax must not exceed GVL.GroupCapacity (set by GroupManager based *)
(*     on healthy units, e.g., opCount * 25). Limits are applied in ReadLimits method. *)
(* 38-177: Device Inputs (20 devices x 7 inputs = 140 indices) *)
(*   - Each device (0-19) has 7 inputs for setpoints, flags, and limits *)
(*   - For devIdx = 0 TO 19, baseIdx = 38 + (devIdx * 7): *)
(*     baseIdx: VoutSetpoint (Voltage setpoint, applied to device in maintenance mode *)
(*              or master in normal mode) *)
(*     baseIdx + 1: IoutSetpoint (Current setpoint, applied to device or master) *)
(*     baseIdx + 2: Flags (WORD, processed in ProcessInputs) *)
(*       - Bit 0 (16#0001): Direction (Forward/reverse) *)
(*       - Bit 1 (16#0002): OperationOn (Operation active) *)
(*       - Bits 2-3 (16#000C): DeviceMode (0-3, e.g., 1 = current mode, 2 = voltage mode) *)
(*       - Bit 4 (16#0010): OutputOn (Device enabled) *)
(*       - Bit 5 (16#0020): OrangeStop *)
(*       - Bit 6 (16#0040): RedStop *)
(*       - Bit 7 (16#0080): EStop *)
(*     baseIdx + 3: VoutSetMin (Minimum voltage limit) *)
(*     baseIdx + 4: VoutSetMax (Maximum voltage limit) *)
(*     baseIdx + 5: IoutSetMin (Minimum current limit) *)
(*     baseIdx + 6: IoutSetMax (Maximum current limit) *)
(*   - Device Index Breakdown (examples): *)
(*     devIdx = 0: 38-44 *)
(*     devIdx = 4: 66-72 *)
(*     devIdx = 19: 171-177 *)
(*   - Note: In normal mode, master device's setpoints/limits are overridden by group *)
(*     inputs (handled in ReadLimits). In maintenance mode, each device uses its own inputs. *)
(* 178+: Unallocated *)
(*      - Available for future expansion *)

(* GVL.NumericOutput Mapping *)
(* Overview: GVL.NumericOutput stores device status, system alarms, group master indices, *)
(* and group capacities. In initialization mode, it handles manufacturer serial data. *)
(* 0-99: Device Outputs (20 devices x 5 outputs = 100 indices) *)
(*   - For devIdx = 0 TO 19, baseIdx = devIdx * 5: *)
(*     baseIdx: Vin (high 16 bits), Vout (low 16 bits) *)
(*     baseIdx + 1: Iout (high), Temperature (low) *)
(*     baseIdx + 2: FanSpeed1 (high), FanSpeed2 (low) *)
(*     baseIdx + 3: FaultStatus (high 16 bits), Status Flags (low bits) *)

(*       - Bit 0: OperationOn *)
(*       - Bit 1: Direction *)
(*       - Bits 2: current*)
(*       - Bits 3: current*)
(*       - Bit 4: OutputOn *)
(*       - Bit 5: OrangeStop *)
(*       - Bit 6: RedStop *)
(*       - Bit 7: EStop *)
(*       - Bit 8: TemperatureFaultHigh *)
(*     baseIdx + 4: FanSpeed1 (high 16 bits) *)
(*   - Example: *)
(*     devIdx = 0: 0-4 *)
(*     devIdx = 4: 20-24 *)
(*     devIdx = 19: 95-99 *)
(* 100: systemAlarms (DWORD, system-wide alarms) *)
(* 101: System Flags (WORD) *)
(*   - Bit 0: GVL.SystemFlags *)
(*   - Bit 1: RefreshTableRequired *)
(*   - Bit 2: GVL.EthercatAliveFromMaster *)
(*   - Bit 3: GVL.RemoteMasterAlive *)
(*   - Bit 4: watchDog (toggled per cycle) *)
(*   - Bit 5: DataRefreshRequired *)
(*   - Bit 6: EL3174_Channel1_Alarm *)
(*   - Bit 7: EL3174_Channel2_Alarm *)
(*   - Bit 8: EL3174_Channel3_Alarm *)
(*   - Bit 9: EL3174_Channel4_Alarm *)
(* 102: GroupMaster[0] (high 16 bits), GroupMaster[1] (low 16 bits) *)
(* 103: GroupMaster[2] (high), GroupMaster[3] (low) *)
(* 104-107: Group Status (outCount high 16 bits, opCount low 16 bits) *)
(*   - 104: LVLA1 (devices 4-7) *)
(*   - 105: LVLA2 (devices 8-11) *)
(*   - 106: LVLA3 (devices 12-15) *)
(*   - 107: LVLA4 (devices 16-19) *)
(*   - outCount: Number of devices with OutputOn *)
(*   - opCount: Number of devices with OperationOn *)
(* 108-111: GVL.GroupCapacity (UINT to DWORD, capacity per group) *)
(*   - 108: LVLA1 *)
(*   - 109: LVLA2 *)
(*   - 110: LVLA3 *)
(*   - 111: LVLA4 *)
(*   - Capacity based on healthy units (opCount * 25), influences group limits *)
(* 0-119 (Initialization Mode): Manufacturer Serial Data *)
(*   - Used for MfrSerialPersistent during initialization cycles *)
(*   - Index calculation: idx = (devIdx * 27) + (i * 3) + j *)
(*   - cmdId (16#80 + i) and serial data packed into WORD *)

METHOD ApplyCommands : BOOL
VAR_INPUT
  devIdx : INT;                            (** Device index **)
  commandCode : UINT;                      (** Command code **)
  data : UINT;                             (** Command data value **)
END_VAR
VAR
  nowTime : TIME;
END_VAR
(** Send CAN commands with polling paused, respecting OutputOn **)
IF devIdx >= 0 AND devIdx <= 19 THEN
  (* Re-arm configuration if communication fault is active for this device. *)
  IF GVL.CommFault[devIdx] THEN
    CanCtrlConfigured[devIdx] := FALSE;
  END_IF;

    (* Ensure CAN control mode is enabled for BIC devices (4..19) only.
      Bus1 DPU devices (0..3) use a different protocol model and should not receive SYSTEM_CONFIG here. *)
  IF (commandCode = 16#0000 OR commandCode = 16#0020 OR commandCode = 16#0030 OR commandCode = 16#0120 OR commandCode = 16#0130)
      AND devIdx >= 4 AND NOT CanCtrlConfigured[devIdx] THEN
    IF fbDeviceManager.WriteDLC4(devIdx, GVL_Constant.CMD_SYSTEM_CONFIG, 16#0005) THEN
      CanCtrlConfigured[devIdx] := TRUE;
    END_IF;
    ApplyCommands := FALSE;
    RETURN;
  END_IF;

  (* DPU manual requires >=50 ms spacing between commands. Apply per-device write pacing globally for safety. *)
  nowTime := TIME();
  IF LastCommandSentTime[devIdx] <> T#0MS AND (nowTime - LastCommandSentTime[devIdx]) < T#50MS THEN
    ApplyCommands := FALSE;
    RETURN;
  END_IF;

  (** Determine command data and clear setpoints based on OutputOn **)
  IF GVL.OutputOn[devIdx] OR commandCode = 16#0000 OR commandCode = 16#0100 THEN
    commandData := data; (** Use provided data for enabled output or non-setpoint commands **)
  ELSE
    commandData := 0; (** Use zero data for setpoint commands if output disabled **)
    (** Clear setpoints for relevant commands **)
    CASE commandCode OF
      16#0020: (** CMD_VOUT_SET **)
        GVL.VoutSetpoint[devIdx] := 0.0; (** Clear forward Vout setpoint **)
      16#0030: (** CMD_IOUT_SET **)
        GVL.IoutSetpoint[devIdx] := 0.0; (** Clear forward Iout setpoint **)
      16#0120: (** CMD_REVERSE_VOUT_SET **)
        GVL.VoutSetRev[devIdx] := 0.0; (** Clear reverse Vout setpoint **)
      16#0130: (** CMD_REVERSE_IOUT_SET **)
        GVL.IoutSetRev[devIdx] := 0.0; (** Clear reverse Iout setpoint **)
    END_CASE;
  END_IF;

  (** Proceed with command **)
  GVL.PollingPaused[devIdx] := TRUE; (** Pause polling for this device **)
  GVL.PollingPauseStartTime[devIdx] := TIME(); (** Record pause start time **)
  GVL.PollingPauseTimeout[devIdx](IN := TRUE, PT := T#100MS); (** Start 100ms timeout **)
  CASE commandCode OF
    16#0000: (** CMD_OPERATION **)
      ApplyCommands := fbDeviceManager.WriteDLC3(devIdx, GVL_Constant.CMD_OPERATION, UINT_TO_BYTE(commandData));
    16#0100: (** CMD_DIRECTION_CTRL **)
      ApplyCommands := fbDeviceManager.WriteDLC3(devIdx, GVL_Constant.CMD_DIRECTION_CTRL, UINT_TO_BYTE(commandData));
    16#0020: (** CMD_VOUT_SET **)
      ApplyCommands := fbDeviceManager.WriteDLC4(devIdx, GVL_Constant.CMD_VOUT_SET, commandData);
    16#0030: (** CMD_IOUT_SET **)
      ApplyCommands := fbDeviceManager.WriteDLC4(devIdx, GVL_Constant.CMD_IOUT_SET, commandData);
    16#0120: (** CMD_REVERSE_VOUT_SET **)
      ApplyCommands := fbDeviceManager.WriteDLC4(devIdx, GVL_Constant.CMD_REVERSE_VOUT_SET, commandData);
    16#0130: (** CMD_REVERSE_IOUT_SET **)
      ApplyCommands := fbDeviceManager.WriteDLC4(devIdx, GVL_Constant.CMD_REVERSE_IOUT_SET, commandData);
    ELSE
      ApplyCommands := FALSE; (** Invalid command code **)
      GVL.PollingPaused[devIdx] := FALSE; (** Resume polling on invalid command **)
      GVL.PollingPauseTimeout[devIdx](IN := FALSE); (** Stop timeout **)
  END_CASE;
  IF ApplyCommands THEN
    LastCommandSentTime[devIdx] := nowTime;
    (* Force immediate feedback polling after setpoint writes. ReadCommands index: 1=VOUT, 2=IOUT *)
    CASE commandCode OF
      16#0020, 16#0120:
        GVL.ReadCommandIndex[devIdx] := 1;
      16#0030, 16#0130:
        GVL.ReadCommandIndex[devIdx] := 2;
    END_CASE;

    GVL.PollingPaused[devIdx] := FALSE; (** Resume polling after successful write **)
    GVL.PollingPauseTimeout[devIdx](IN := FALSE); (** Stop timeout **)
  END_IF;
ELSE
  ApplyCommands := FALSE; (** Invalid device index **)
END_IF;
END_METHOD

METHOD ProcessInputs
VAR
  devIdx : INT;                            (** Device index **)
  baseIdx : INT;                           (** Base index for device inputs **)
  flags : WORD;                            (** Device-specific input flags **)
  systemFlags : WORD;                      (** System flags **)
  safetyOK : BOOL;                         (** Safety status **)
  groupIdx : INT;                          (** Group index **)
  memberIdx : INT;                         (** Member device index **)
  masterIdx : INT;                         (** Master device index **)
  groupBase : INT;                         (** Base index for group devices **)
  maintenanceMode : BOOL;                  (** Maintenance mode status **)
  isGroupMaster : BOOL;                    (** Group master flag **)
  clampedVout : UINT;                      (** Clamped voltage setpoint **)
  clampedIout : UINT;                      (** Clamped current setpoint **)
  i : INT;                                 (** Loop index for channel mapping **)
  factorNibble : UINT;                     (** Factor nibble from scaling-factor fields **)
  setpointIout : REAL;                     (** Clamped Iout setpoint before scaling **)
  setpointVout : REAL;                     (** Clamped Vout setpoint before scaling **)
	j: INT;
END_VAR


(** Comment Section: GVL.NumericInput Mapping for ProcessInputs **)
(** This method processes system, group, and device inputs from GVL.NumericInput, setting **)
(** setpoints, flags, and maintenance mode. In normal mode (maintenanceMode = FALSE), **)
(** group flags (Direction, OperationOn, OutputOn) are set for all devices in the group **)
(** (4-19), but DeviceMode (Voltage, Current, Standby) and setpoints (VoutSetpoint, **)
(** IoutSetpoint) are set only for the group master. In maintenance mode or for devices **)
(** 0-3, all flags and setpoints are set per device. Group limits are applied to all **)
(** devices in the group, with IoutSetMax constrained by the minimum of GroupIoutSetMax **)
(** and GVL.GroupCapacity (set by GroupManager.UpdateGroupCapacity using input voltage **)
(** feedback, GVL.Vin > 100). GroupMaster is updated by GroupManager.UpdateGroupMasters **)
(** using input voltage feedback. Groups: 0=4-7, 1=8-11, 2=12-15, 3=16-19. **)
(** Flags for groups and devices use identical bit assignments. **)

(** GVL.NumericInput Mapping **)
(** 0-4: System-Level Inputs **)
(**   0: GVL.SystemAlarms (WORD to UINT) **)
(**      - System-wide alarms, read into GVL.SystemAlarms **)
(**   1: System Flags (WORD) **)
(**      - Bit 0 (16#0001): GVL.SystemFlags (sets maintenanceMode) **)
(**      - Bit 1 (16#0002): GVL.EthercatAliveFromMaster **)
(**      - Bit 2 (16#0004): GVL.RemoteMasterAlive **)
(**   2: Morphee Initialization Signal **)
(**      - Used in UpdateOutputs, not processed here **)
(**   3-4: Reserved **)
(** 5-9: Unallocated **)
(** 10-37: Group Inputs (4 groups x 7 inputs) **)
(**   - For groupIdx = 0 TO 3, baseIdx = 10 + (groupIdx * 7): **)
(**     baseIdx: GroupVoutSetpoint **)
(**     baseIdx + 1: GroupIoutSetpoint **)
(**     baseIdx + 2: Group Flags **)
(**       - Bit 0 (16#0001): Direction **)
(**       - Bit 1 (16#0002): OperationOn **)
(**       - Bit 2 (16#0004): DeviceMode Current **)
(**       - Bit 3 (16#0008): DeviceMode Voltage **)
(**       - Bit 4 (16#0010): OutputOn **)
(**     baseIdx + 3: GroupVoutSetMin **)
(**     baseIdx + 4: GroupVoutSetMax **)
(**     baseIdx + 5: GroupIoutSetMin **)
(**     baseIdx + 6: GroupIoutSetMax **)
(**   - GroupVoutSetpoint, GroupIoutSetpoint, and DeviceMode applied to master device only in normal mode **)
(**   - GroupVoutSetMin, GroupVoutSetMax, GroupIoutSetMin, GroupIoutSetMax applied to all devices in group **)
(**   - Group Flags (Direction, OperationOn, OutputOn) set for all devices in group in normal mode **)
(** 38-177: Device Inputs (20 devices x 7 inputs) **)
(**   - For devIdx = 0 TO 19, baseIdx = 38 + (devIdx * 7): **)
(**     baseIdx: VoutSetpoint (Read here) **)
(**     baseIdx + 1: IoutSetpoint (Read here) **)
(**     baseIdx + 2: Flags (Read here) **)
(**       - Bit 0 (16#0001): Direction **)
(**       - Bit 1 (16#0002): OperationOn **)
(**       - Bit 2 (16#0004): DeviceMode Current **)
(**       - Bit 3 (16#0008): DeviceMode Voltage **)
(**       - Bit 4 (16#0010): OutputOn **)
(**       - Bit 5 (16#0020): OrangeStop **)
(**       - Bit 6 (16#0040): RedStop **)
(**       - Bit 7 (16#0080): EStop **)
(**     baseIdx + 3: VoutSetMin (Set in ReadLimits) **)
(**     baseIdx + 4: VoutSetMax **)
(**     baseIdx + 5: IoutSetMin **)
(**     baseIdx + 6: IoutSetMax **)
(** 178+: Unallocated **)

(** Read limits first **)
THIS^.ReadLimits();

(** Read system alarms **)
GVL.SystemAlarms := GVL.NumericInput[0]; (** Index 0: System alarms **)

(** Read system flags **)
systemFlags := GVL.NumericInput[1]; (** Index 1: System flags **)
GVL.SystemFlags := TO_BYTE(systemFlags AND 16#0001);
GVL.EthercatAliveFromMaster := (systemFlags AND 16#0002) <> 0;
GVL.RemoteMasterAlive := (systemFlags AND 16#0004) <> 0;
maintenanceMode := (systemFlags AND 16#0001) <> 0; (** Maintenance mode flag **)

(** Process EL2809 and EL2798 inputs **)
FOR j:=0 TO 2 DO
GVL.EL2809_InputFlags[j] := GVL.NumericInput[5+j]; (** Index 5: EL2809 flags **)
	FOR i := 0 TO 15 DO
	  GVL.EL2809_Output[j,i] := (GVL.EL2809_InputFlags[j] AND SHL(TO_WORD(1), i)) <> 0;
	END_FOR;
END_FOR;

GVL.EL2798_InputFlags := TO_BYTE(GVL.NumericInput[6]); (** Index 6: EL2798 flags **)
FOR i := 0 TO 7 DO
  GVL.EL2798_Output[i] := (GVL.EL2798_InputFlags AND SHL(TO_BYTE(1), i)) <> 0;
END_FOR;

(** Process group inputs for 4 groups **)
FOR groupIdx := 0 TO 3 DO
  baseIdx := 10 + (groupIdx * 7); (** Group inputs start at 10 **)
  
  (** Read group inputs **)
  IF baseIdx + 6 < SIZEOF(GVL.NumericInput) / SIZEOF(GVL.NumericInput[0]) THEN
    (** Read master setpoints/flags from temp test input when enabled, else from live NumericInput **)
    IF GVL.UseTempGroupInputs AND (baseIdx - 10) + 6 < SIZEOF(GVL.TempGroupInput) / SIZEOF(GVL.TempGroupInput[0]) THEN
      setpointVout := UINT_TO_REAL(GVL.TempGroupInput[baseIdx - 10]);
      setpointIout := UINT_TO_REAL(GVL.TempGroupInput[(baseIdx - 10) + 1]);
      flags := GVL.TempGroupInput[(baseIdx - 10) + 2];
    ELSE
      setpointVout := UINT_TO_REAL(GVL.NumericInput[baseIdx]);
      setpointIout := UINT_TO_REAL(GVL.NumericInput[baseIdx + 1]);
      flags := GVL.NumericInput[baseIdx + 2];
    END_IF;
    
    (** Identify master device for the group **)
    masterIdx := GVL.GroupMaster[groupIdx]; (** Use GVL.GroupMaster for master device index **)
    
    (** Apply setpoints and DeviceMode to master device in normal mode **)
    IF NOT maintenanceMode AND masterIdx >= 4 AND masterIdx <= 19 THEN
      (** Set DeviceMode for master **)
      GVL.Voltage[masterIdx] := (flags AND 16#0008) <> 0;     (** Bit 3: DeviceMode Voltage **)
      GVL.Current[masterIdx] := (flags AND 16#0004) <> 0;     (** Bit 2: DeviceMode Current **)
      GVL.Standby[masterIdx] := NOT (GVL.Voltage[masterIdx] OR GVL.Current[masterIdx]); (** Standby when neither Voltage nor Current **)

      (** Set OutputOn for master BEFORE sending setpoint so ApplyCommands guard uses current value **)
      (** Also reset last setpoint cache when OutputOn transitions FALSE->TRUE to force resend **)
      IF (flags AND 16#0010) <> 0 AND NOT GVL.OutputOn[masterIdx] THEN
        THIS^.LastVoutSetpoint[masterIdx] := 0;
        THIS^.LastIoutSetpoint[masterIdx] := 0;
      END_IF;
      GVL.OutputOn[masterIdx] := (flags AND 16#0010) <> 0;

      (** Clamp setpoints within group limits **)
      IF GVL.UseTempGroupInputs AND (baseIdx - 10) + 6 < SIZEOF(GVL.TempGroupInput) / SIZEOF(GVL.TempGroupInput[0]) THEN
        setpointVout := MIN(MAX(setpointVout / 100, UINT_TO_REAL(GVL.TempGroupInput[(baseIdx - 10) + 3])), UINT_TO_REAL(GVL.TempGroupInput[(baseIdx - 10) + 4]));
        setpointIout := MIN(MAX(setpointIout / 100, UINT_TO_REAL(GVL.TempGroupInput[(baseIdx - 10) + 5])), UINT_TO_REAL(MIN(GVL.TempGroupInput[(baseIdx - 10) + 6], GVL.GroupCapacity[groupIdx])));
      ELSE
        setpointVout := MIN(MAX(setpointVout / 100, UINT_TO_REAL(GVL.NumericInput[baseIdx + 3])), UINT_TO_REAL(GVL.NumericInput[baseIdx + 4])); (** Clamp Vout to GroupVoutSetMin/Max **)
        setpointIout := MIN(MAX(setpointIout / 100, UINT_TO_REAL(GVL.NumericInput[baseIdx + 5])), UINT_TO_REAL(MIN(GVL.NumericInput[baseIdx + 6], GVL.GroupCapacity[groupIdx]))); (** Clamp Iout to GroupIoutSetMin/min(GroupIoutSetMax, GroupCapacity) **)
      END_IF;
      
      (** Scale and apply to master **)
      clampedVout := REAL_TO_UINT(setpointVout * 100.0);
      clampedIout := REAL_TO_UINT(setpointIout * 100.0);
      
      IF clampedVout <> THIS^.LastVoutSetpoint[masterIdx] THEN
        IF THIS^.ApplyCommands(masterIdx, GVL_Constant.CMD_VOUT_SET, clampedVout) THEN (** CMD_VOUT_SET **)
          THIS^.LastVoutSetpoint[masterIdx] := clampedVout;
        END_IF;
      END_IF;
      
      IF clampedIout <> THIS^.LastIoutSetpoint[masterIdx] THEN
        IF THIS^.ApplyCommands(masterIdx, GVL_Constant.CMD_IOUT_SET, clampedIout) THEN (** CMD_IOUT_SET **)
          THIS^.LastIoutSetpoint[masterIdx] := clampedIout;
        END_IF;
      END_IF;
    END_IF;
    
    (** Set group flags (excluding DeviceMode) and limits for all devices in group in normal mode **)
    IF NOT maintenanceMode THEN
      FOR devIdx := 0 TO 19 DO
        IF GVL.GroupMembership[devIdx] = groupIdx THEN
          (** Set group flags **)
          GVL.Direction[devIdx] := (flags AND 16#0001) <> 0;   (** Bit 0: Direction **)
          GVL.OperationOn[devIdx] := (flags AND 16#0002) <> 0; (** Bit 1: OperationOn **)
          GVL.OutputOn[devIdx] := (flags AND 16#0010) <> 0;    (** Bit 4: OutputOn **)
          
